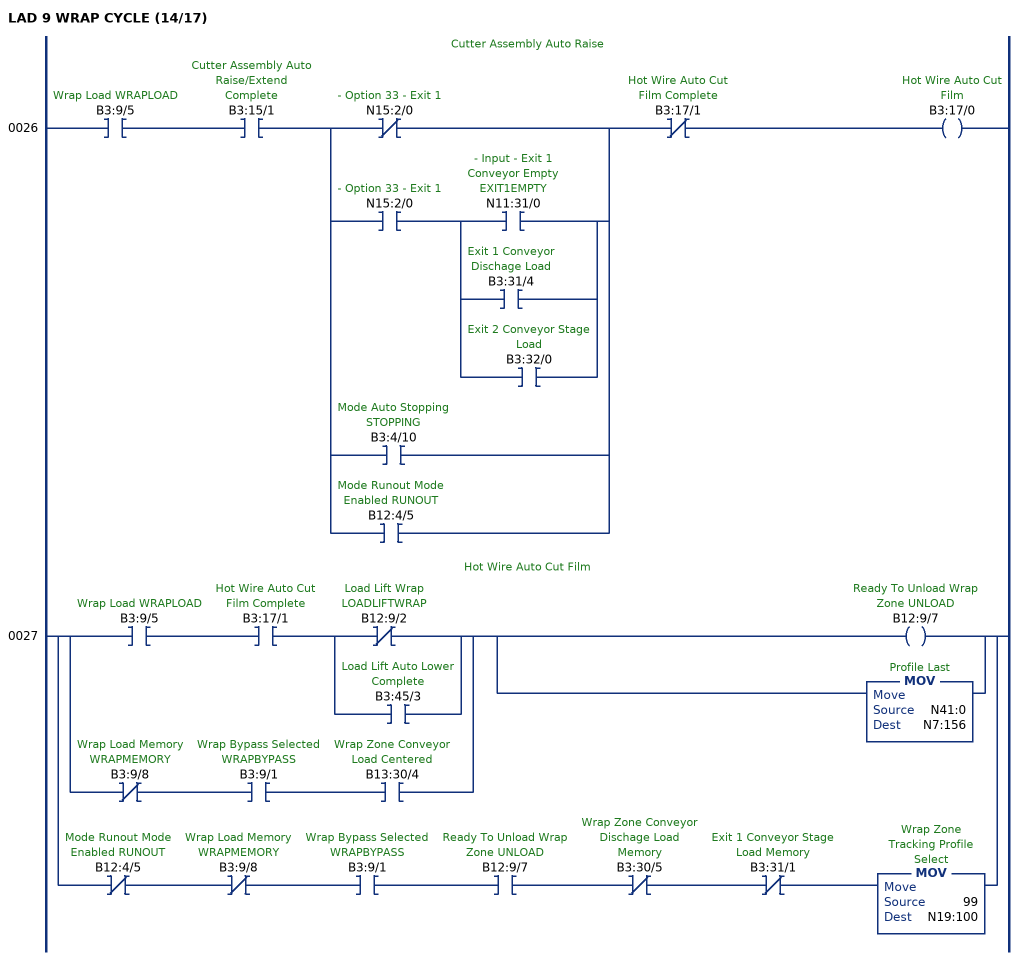
% Rung: 26 %
% Cutter Assembly Auto Raise %
SOR XIC B3:9/5 XIC B3:15/1 BST XIO N15:2/0 NXB XIC N15:2/0 BST XIC N11:31/0 NXB XIC B3:31/4 NXB XIC B3:32/0 BND NXB XIC B3:4/10 NXB XIC B12:4/5 BND XIO B3:17/1 OTE B3:17/0 EOR
%   B3:9/5  WRAPLOAD  "Wrap Load" %
%   B3:15/1  "Cutter Assembly Auto Raise/Extend Complete" %
%   N15:2/0  "- Option 33 - Exit 1" %
%   N11:31/0  EXIT1EMPTY  "- Input - Exit 1 Conveyor Empty" %
%   B3:31/4  "Exit 1 Conveyor Dischage Load" %
%   B3:32/0  "Exit 2 Conveyor Stage Load" %
%   B3:4/10  STOPPING  "Mode Auto Stopping" %
%   B12:4/5  RUNOUT  "Mode Runout Mode Enabled" %
%   B3:17/1  "Hot Wire Auto Cut Film Complete" %
%   B3:17/0  "Hot Wire Auto Cut Film" %
% Rung: 27 %
% Hot Wire Auto Cut Film %
SOR BST BST XIC B3:9/5 XIC B3:17/1 BST XIO B12:9/2 NXB XIC B3:45/3 BND NXB XIO B3:9/8 XIC B3:9/1 XIC B13:30/4 BND BST OTE B12:9/7 NXB MOV N41:0 N7:156 BND NXB XIO B12:4/5 XIO B3:9/8 XIC B3:9/1 XIC B12:9/7 XIO B3:30/5 XIO B3:31/1 MOV 99 N19:100 BND EOR
%   B3:9/5  WRAPLOAD  "Wrap Load" %
%   B3:17/1  "Hot Wire Auto Cut Film Complete" %
%   B12:9/2  LOADLIFTWRAP  "Load Lift Wrap" %
%   B3:45/3  "Load Lift Auto Lower Complete" %
%   B3:9/8  WRAPMEMORY  "Wrap Load Memory" %
%   B3:9/1  WRAPBYPASS  "Wrap Bypass Selected" %
%   B13:30/4  "Wrap Zone Conveyor Load Centered" %
%   B12:9/7  UNLOAD  "Ready To Unload Wrap Zone" %
%   N41:0  "Profile Max Index" %
%   N7:156  "Profile Last" %
%   B12:4/5  RUNOUT  "Mode Runout Mode Enabled" %
%   B3:30/5  "Wrap Zone Conveyor Dischage Load Memory" %
%   B3:31/1  "Exit 1 Conveyor Stage Load Memory" %
%   N19:100  "Wrap Zone Tracking Profile Select" %

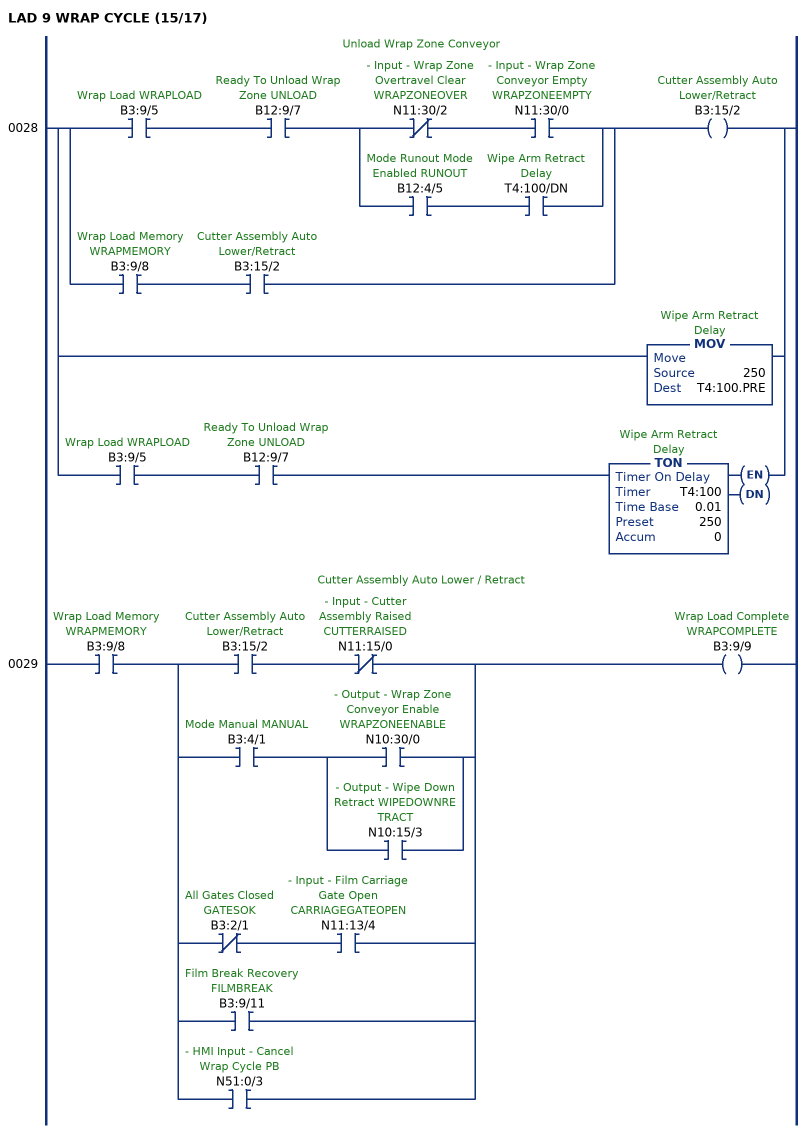
% Rung: 28 %
% Unload Wrap Zone Conveyor %
SOR BST BST XIC B3:9/5 XIC B12:9/7 BST XIO N11:30/2 XIC N11:30/0 NXB XIC B12:4/5 XIC T4:100/DN BND NXB XIC B3:9/8 XIC B3:15/2 BND OTE B3:15/2 NXB MOV 250 T4:100.PRE NXB XIC B3:9/5 XIC B12:9/7 TON T4:100 0.01 250 0 BND EOR
%   B3:9/5  WRAPLOAD  "Wrap Load" %
%   B12:9/7  UNLOAD  "Ready To Unload Wrap Zone" %
%   N11:30/2  WRAPZONEOVER  "- Input - Wrap Zone Overtravel Clear" %
%   N11:30/0  WRAPZONEEMPTY  "- Input - Wrap Zone Conveyor Empty" %
%   B12:4/5  RUNOUT  "Mode Runout Mode Enabled" %
%   T4:100  "Wipe Arm Retract Delay" %
%   B3:9/8  WRAPMEMORY  "Wrap Load Memory" %
%   B3:15/2  "Cutter Assembly Auto Lower/Retract" %
% Rung: 29 %
% Cutter Assembly Auto Lower / Retract %
SOR XIC B3:9/8 BST XIC B3:15/2 XIO N11:15/0 NXB XIC B3:4/1 BST XIC N10:30/0 NXB XIC N10:15/3 BND NXB XIO B3:2/1 XIC N11:13/4 NXB XIC B3:9/11 NXB XIC N51:0/3 BND OTE B3:9/9 EOR
%   B3:9/8  WRAPMEMORY  "Wrap Load Memory" %
%   B3:15/2  "Cutter Assembly Auto Lower/Retract" %
%   N11:15/0  CUTTERRAISED  "- Input - Cutter Assembly Raised" %
%   B3:4/1  MANUAL  "Mode Manual" %
%   N10:30/0  WRAPZONEENABLE  "- Output - Wrap Zone Conveyor Enable" %
%   N10:15/3  WIPEDOWNRETRACT  "- Output - Wipe Down Retract" %
%   B3:2/1  GATESOK  "All Gates Closed" %
%   N11:13/4  CARRIAGEGATEOPEN  "- Input - Film Carriage Gate Open" %
%   B3:9/11  FILMBREAK  "Film Break Recovery" %
%   N51:0/3  "- HMI Input - Cancel Wrap Cycle PB" %
%   B3:9/9  WRAPCOMPLETE  "Wrap Load Complete" %

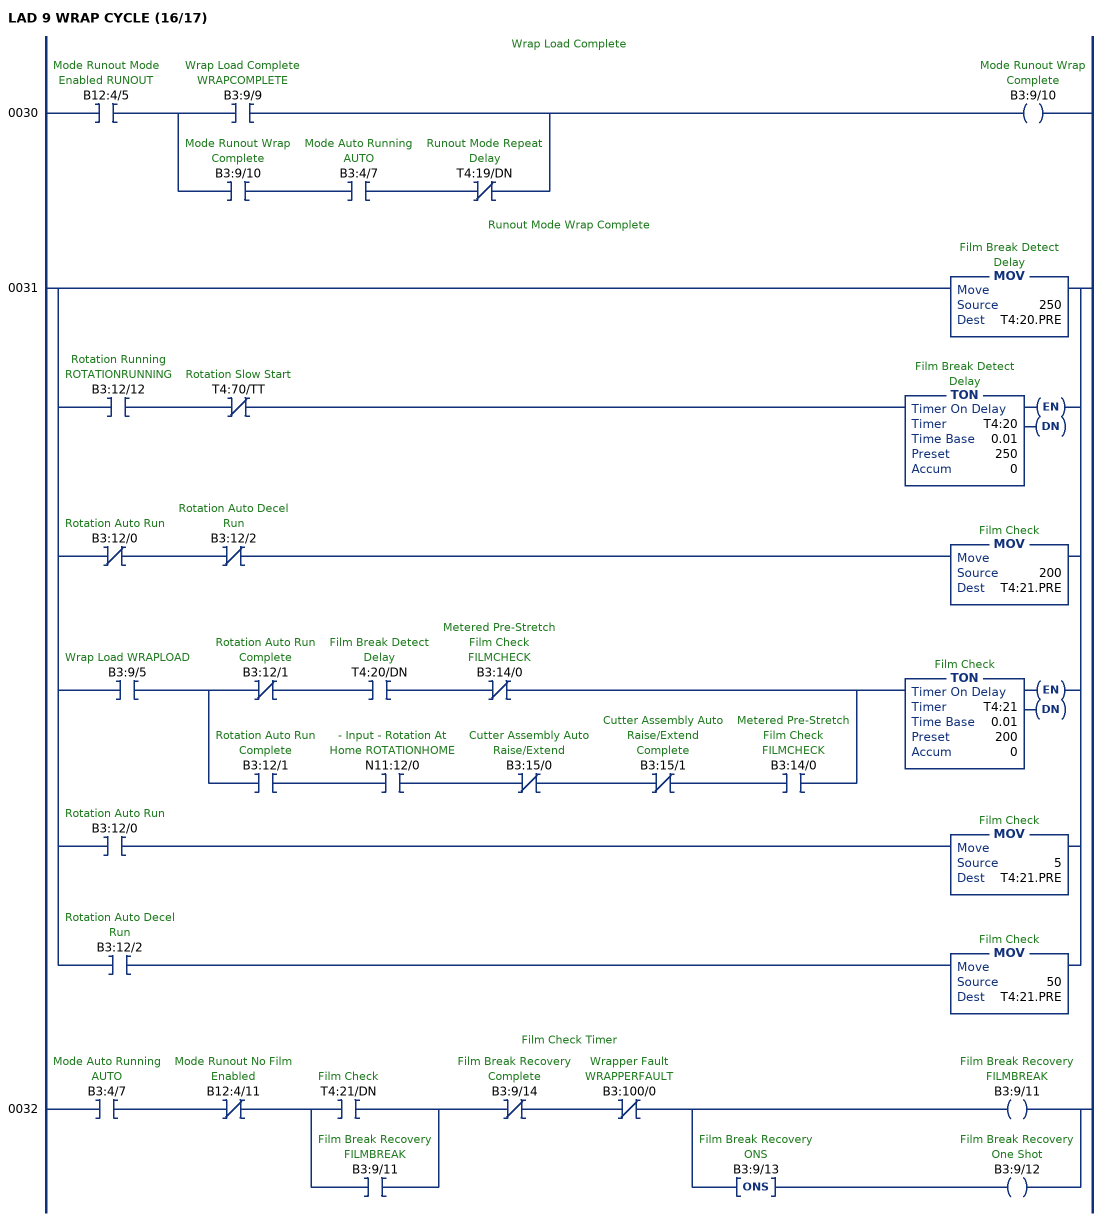
% Rung: 30 %
% Wrap Load Complete %
SOR XIC B12:4/5 BST XIC B3:9/9 NXB XIC B3:9/10 XIC B3:4/7 XIO T4:19/DN BND OTE B3:9/10 EOR
%   B12:4/5  RUNOUT  "Mode Runout Mode Enabled" %
%   B3:9/9  WRAPCOMPLETE  "Wrap Load Complete" %
%   B3:9/10  "Mode Runout Wrap Complete" %
%   B3:4/7  AUTO  "Mode Auto Running" %
%   T4:19  "Runout Mode Repeat Delay" %
% Rung: 31 %
% Runout Mode Wrap Complete %
SOR BST MOV 250 T4:20.PRE NXB XIC B3:12/12 XIO T4:70/TT TON T4:20 0.01 250 0 NXB XIO B3:12/0 XIO B3:12/2 MOV 200 T4:21.PRE NXB XIC B3:9/5 BST XIO B3:12/1 XIC T4:20/DN XIO B3:14/0 NXB XIC B3:12/1 XIC N11:12/0 XIO B3:15/0 XIO B3:15/1 XIC B3:14/0 BND TON T4:21 0.01 200 0 NXB BST XIC B3:12/0 MOV 5 T4:21.PRE NXB XIC B3:12/2 MOV 50 T4:21.PRE BND BND EOR
%   T4:20  "Film Break Detect Delay" %
%   B3:12/12  ROTATIONRUNNING  "Rotation Running" %
%   T4:70  "Rotation Slow Start" %
%   B3:12/0  "Rotation Auto Run" %
%   B3:12/2  "Rotation Auto Decel Run" %
%   T4:21  "Film Check" %
%   B3:9/5  WRAPLOAD  "Wrap Load" %
%   B3:12/1  "Rotation Auto Run Complete" %
%   B3:14/0  FILMCHECK  "Metered Pre-Stretch Film Check" %
%   N11:12/0  ROTATIONHOME  "- Input - Rotation At Home" %
%   B3:15/0  "Cutter Assembly Auto Raise/Extend" %
%   B3:15/1  "Cutter Assembly Auto Raise/Extend Complete" %
% Rung: 32 %
% Film Check Timer %
SOR XIC B3:4/7 XIO B12:4/11 BST XIC T4:21/DN NXB XIC B3:9/11 BND XIO B3:9/14 XIO B3:100/0 BST OTE B3:9/11 NXB ONS B3:9/13 OTE B3:9/12 BND EOR
%   B3:4/7  AUTO  "Mode Auto Running" %
%   B12:4/11  "Mode Runout No Film Enabled" %
%   T4:21  "Film Check" %
%   B3:9/11  FILMBREAK  "Film Break Recovery" %
%   B3:9/14  "Film Break Recovery Complete" %
%   B3:100/0  WRAPPERFAULT  "Wrapper Fault" %
%   B3:9/13  "Film Break Recovery ONS" %
%   B3:9/12  "Film Break Recovery One Shot" %

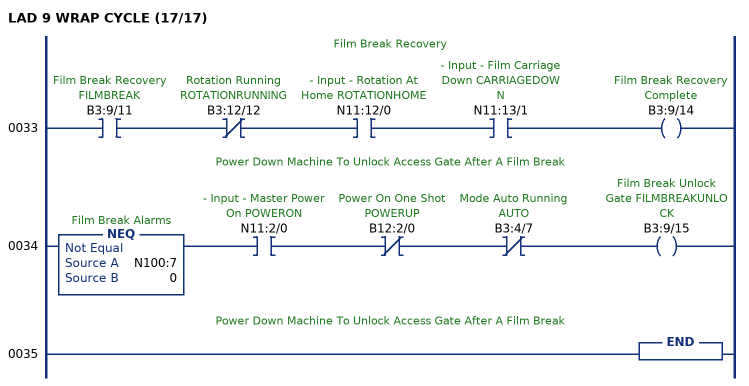
% Rung: 33 %
% Film Break Recovery %
SOR XIC B3:9/11 XIO B3:12/12 XIC N11:12/0 XIC N11:13/1 OTE B3:9/14 EOR
%   B3:9/11  FILMBREAK  "Film Break Recovery" %
%   B3:12/12  ROTATIONRUNNING  "Rotation Running" %
%   N11:12/0  ROTATIONHOME  "- Input - Rotation At Home" %
%   N11:13/1  CARRIAGEDOWN  "- Input - Film Carriage Down" %
%   B3:9/14  "Film Break Recovery Complete" %
% Rung: 34 %
% Power Down Machine To Unlock Access Gate After A Film Break %
SOR NEQ N100:7 0 XIC N11:2/0 XIO B12:2/0 XIO B3:4/7 OTE B3:9/15 EOR
%   N100:7  "Film Break Alarms" %
%   N11:2/0  POWERON  "- Input - Master Power On" %
%   B12:2/0  POWERUP  "Power On One Shot" %
%   B3:4/7  AUTO  "Mode Auto Running" %
%   B3:9/15  FILMBREAKUNLOCK  "Film Break Unlock Gate" %
% Rung: 35 %
% Power Down Machine To Unlock Access Gate After A Film Break %
SOR END EOR

LADDER 10 "OUTPUTS"
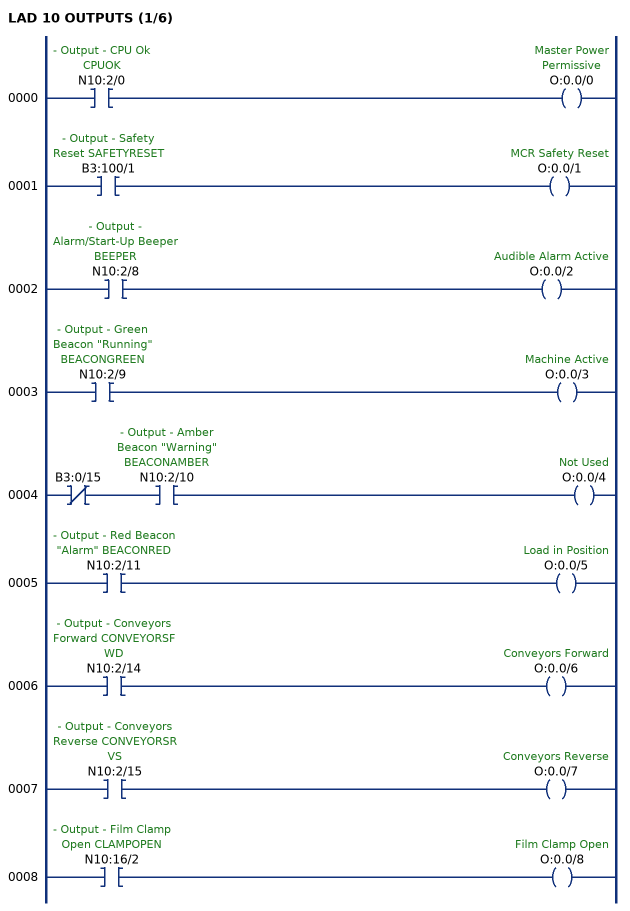
% Rung: 0 %
SOR XIC N10:2/0 OTE O:0.0/0 EOR
%   N10:2/0  CPUOK  "- Output - CPU Ok" %
%   O:0.0/0  "Master Power Permissive" %
% Rung: 1 %
SOR XIC B3:100/1 OTE O:0.0/1 EOR
%   B3:100/1  SAFETYRESET  "- Output - Safety Reset" %
%   O:0.0/1  "MCR Safety Reset" %
% Rung: 2 %
SOR XIC N10:2/8 OTE O:0.0/2 EOR
%   N10:2/8  BEEPER  "- Output - Alarm/Start-Up Beeper" %
%   O:0.0/2  "Audible Alarm Active" %
% Rung: 3 %
SOR XIC N10:2/9 OTE O:0.0/3 EOR
%   N10:2/9  BEACONGREEN  "- Output - Green Beacon "Running"" %
%   O:0.0/3  "Machine Active" %
% Rung: 4 %
SOR XIO B3:0/15 XIC N10:2/10 OTE O:0.0/4 EOR
%   N10:2/10  BEACONAMBER  "- Output - Amber Beacon "Warning"" %
%   O:0.0/4  "Not Used" %
% Rung: 5 %
SOR XIC N10:2/11 OTE O:0.0/5 EOR
%   N10:2/11  BEACONRED  "- Output - Red Beacon "Alarm"" %
%   O:0.0/5  "Load in Position" %
% Rung: 6 %
SOR XIC N10:2/14 OTE O:0.0/6 EOR
%   N10:2/14  CONVEYORSFWD  "- Output - Conveyors Forward" %
%   O:0.0/6  "Conveyors Forward" %
% Rung: 7 %
SOR XIC N10:2/15 OTE O:0.0/7 EOR
%   N10:2/15  CONVEYORSRVS  "- Output - Conveyors Reverse" %
%   O:0.0/7  "Conveyors Reverse" %
% Rung: 8 %
SOR XIC N10:16/2 OTE O:0.0/8 EOR
%   N10:16/2  CLAMPOPEN  "- Output - Film Clamp Open" %
%   O:0.0/8  "Film Clamp Open" %

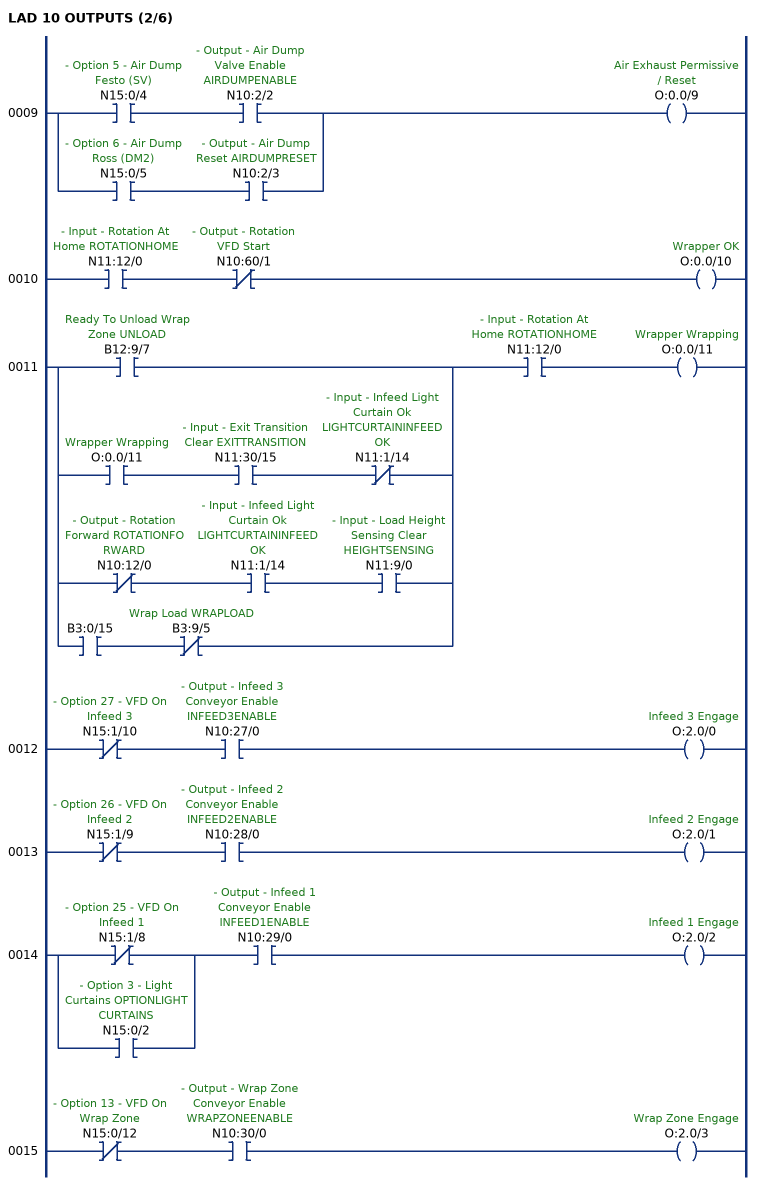
% Rung: 9 %
SOR BST XIC N15:0/4 XIC N10:2/2 NXB XIC N15:0/5 XIC N10:2/3 BND OTE O:0.0/9 EOR
%   N15:0/4  "- Option 5 - Air Dump Festo (SV)" %
%   N10:2/2  AIRDUMPENABLE  "- Output - Air Dump Valve Enable" %
%   N15:0/5  "- Option 6 - Air Dump Ross (DM2)" %
%   N10:2/3  AIRDUMPRESET  "- Output - Air Dump Reset" %
%   O:0.0/9  "Air Exhaust Permissive / Reset" %
% Rung: 10 %
SOR XIC N11:12/0 XIO N10:60/1 OTE O:0.0/10 EOR
%   N11:12/0  ROTATIONHOME  "- Input - Rotation At Home" %
%   N10:60/1  "- Output - Rotation VFD Start" %
%   O:0.0/10  "Wrapper OK" %
% Rung: 11 %
SOR BST XIC B12:9/7 NXB BST XIC O:0.0/11 XIC N11:30/15 XIO N11:1/14 NXB XIO N10:12/0 XIC N11:1/14 XIC N11:9/0 BND NXB XIC B3:0/15 XIO B3:9/5 BND XIC N11:12/0 OTE O:0.0/11 EOR
%   B12:9/7  UNLOAD  "Ready To Unload Wrap Zone" %
%   O:0.0/11  "Wrapper Wrapping" %
%   N11:30/15  EXITTRANSITION  "- Input - Exit Transition Clear" %
%   N11:1/14  LIGHTCURTAININFEEDOK  "- Input - Infeed Light Curtain Ok" %
%   N10:12/0  ROTATIONFORWARD  "- Output - Rotation Forward" %
%   N11:9/0  HEIGHTSENSING  "- Input - Load Height Sensing Clear" %
%   B3:9/5  WRAPLOAD  "Wrap Load" %
%   N11:12/0  ROTATIONHOME  "- Input - Rotation At Home" %
% Rung: 12 %
SOR XIO N15:1/10 XIC N10:27/0 OTE O:2.0/0 EOR
%   N15:1/10  "- Option 27 - VFD On Infeed 3" %
%   N10:27/0  INFEED3ENABLE  "- Output - Infeed 3 Conveyor Enable" %
%   O:2.0/0  "Infeed 3 Engage" %
% Rung: 13 %
SOR XIO N15:1/9 XIC N10:28/0 OTE O:2.0/1 EOR
%   N15:1/9  "- Option 26 - VFD On Infeed 2" %
%   N10:28/0  INFEED2ENABLE  "- Output - Infeed 2 Conveyor Enable" %
%   O:2.0/1  "Infeed 2 Engage" %
% Rung: 14 %
SOR BST XIO N15:1/8 NXB XIC N15:0/2 BND XIC N10:29/0 OTE O:2.0/2 EOR
%   N15:1/8  "- Option 25 - VFD On Infeed 1" %
%   N15:0/2  OPTIONLIGHTCURTAINS  "- Option 3 - Light Curtains" %
%   N10:29/0  INFEED1ENABLE  "- Output - Infeed 1 Conveyor Enable" %
%   O:2.0/2  "Infeed 1 Engage" %
% Rung: 15 %
SOR XIO N15:0/12 XIC N10:30/0 OTE O:2.0/3 EOR
%   N15:0/12  "- Option 13 - VFD On Wrap Zone" %
%   N10:30/0  WRAPZONEENABLE  "- Output - Wrap Zone Conveyor Enable" %
%   O:2.0/3  "Wrap Zone Engage" %

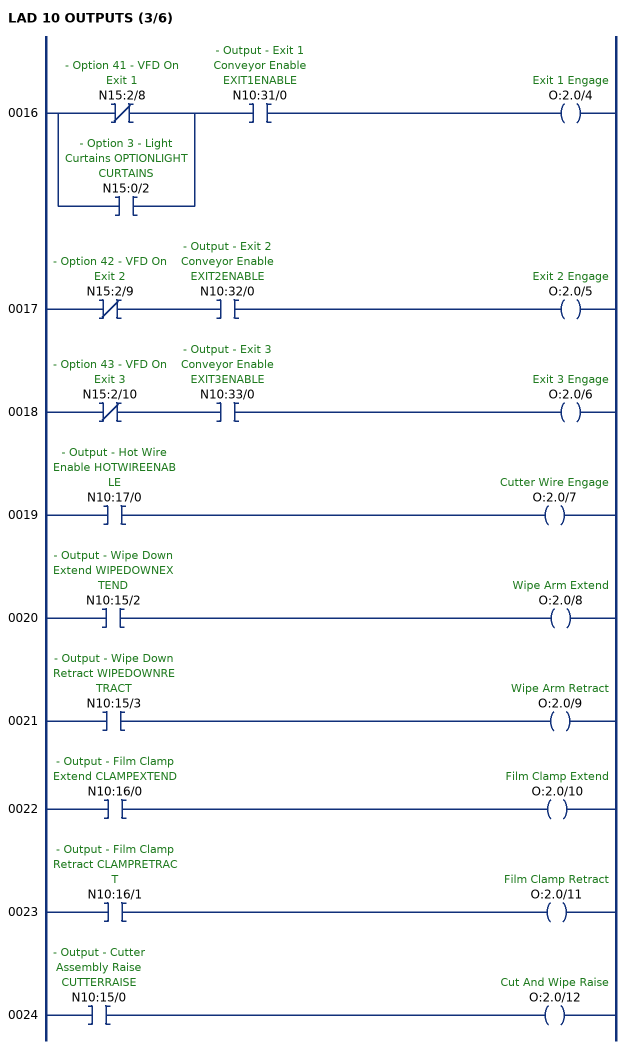
% Rung: 16 %
SOR BST XIO N15:2/8 NXB XIC N15:0/2 BND XIC N10:31/0 OTE O:2.0/4 EOR
%   N15:2/8  "- Option 41 - VFD On Exit 1" %
%   N15:0/2  OPTIONLIGHTCURTAINS  "- Option 3 - Light Curtains" %
%   N10:31/0  EXIT1ENABLE  "- Output - Exit 1 Conveyor Enable" %
%   O:2.0/4  "Exit 1 Engage" %
% Rung: 17 %
SOR XIO N15:2/9 XIC N10:32/0 OTE O:2.0/5 EOR
%   N15:2/9  "- Option 42 - VFD On Exit 2" %
%   N10:32/0  EXIT2ENABLE  "- Output - Exit 2 Conveyor Enable" %
%   O:2.0/5  "Exit 2 Engage" %
% Rung: 18 %
SOR XIO N15:2/10 XIC N10:33/0 OTE O:2.0/6 EOR
%   N15:2/10  "- Option 43 - VFD On Exit 3" %
%   N10:33/0  EXIT3ENABLE  "- Output - Exit 3 Conveyor Enable" %
%   O:2.0/6  "Exit 3 Engage" %
% Rung: 19 %
SOR XIC N10:17/0 OTE O:2.0/7 EOR
%   N10:17/0  HOTWIREENABLE  "- Output - Hot Wire Enable" %
%   O:2.0/7  "Cutter Wire Engage" %
% Rung: 20 %
SOR XIC N10:15/2 OTE O:2.0/8 EOR
%   N10:15/2  WIPEDOWNEXTEND  "- Output - Wipe Down Extend" %
%   O:2.0/8  "Wipe Arm Extend" %
% Rung: 21 %
SOR XIC N10:15/3 OTE O:2.0/9 EOR
%   N10:15/3  WIPEDOWNRETRACT  "- Output - Wipe Down Retract" %
%   O:2.0/9  "Wipe Arm Retract" %
% Rung: 22 %
SOR XIC N10:16/0 OTE O:2.0/10 EOR
%   N10:16/0  CLAMPEXTEND  "- Output - Film Clamp Extend" %
%   O:2.0/10  "Film Clamp Extend" %
% Rung: 23 %
SOR XIC N10:16/1 OTE O:2.0/11 EOR
%   N10:16/1  CLAMPRETRACT  "- Output - Film Clamp Retract" %
%   O:2.0/11  "Film Clamp Retract" %
% Rung: 24 %
SOR XIC N10:15/0 OTE O:2.0/12 EOR
%   N10:15/0  CUTTERRAISE  "- Output - Cutter Assembly Raise" %
%   O:2.0/12  "Cut And Wipe Raise" %

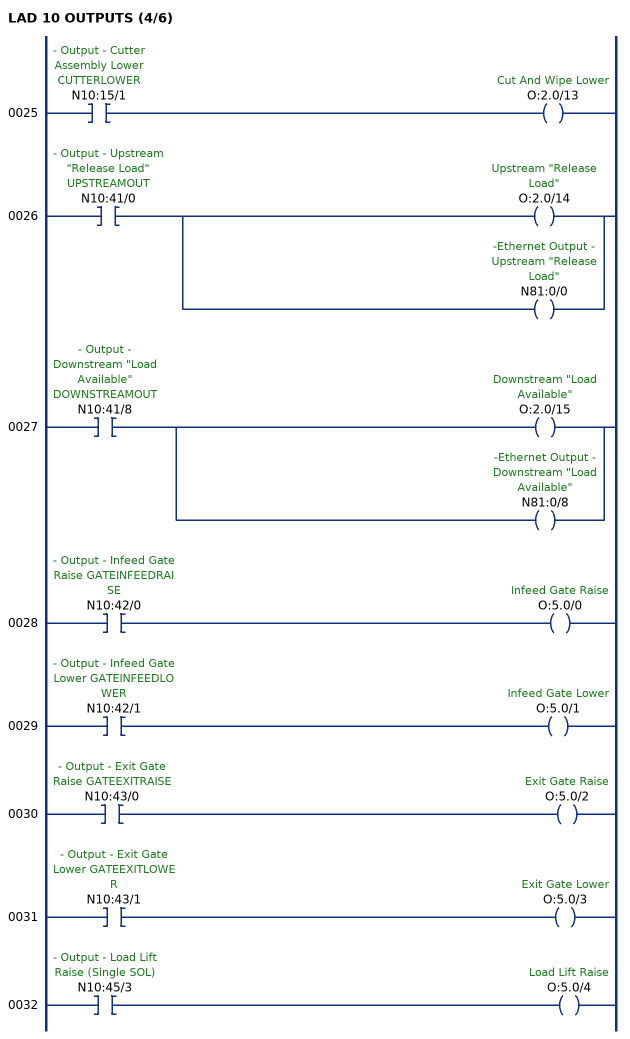
% Rung: 25 %
SOR XIC N10:15/1 OTE O:2.0/13 EOR
%   N10:15/1  CUTTERLOWER  "- Output - Cutter Assembly Lower" %
%   O:2.0/13  "Cut And Wipe Lower" %
% Rung: 26 %
SOR XIC N10:41/0 BST OTE O:2.0/14 NXB OTE N81:0/0 BND EOR
%   N10:41/0  UPSTREAMOUT  "- Output - Upstream "Release Load"" %
%   O:2.0/14  "Upstream "Release Load"" %
%   N81:0/0  "-Ethernet Output - Upstream "Release Load"" %
% Rung: 27 %
SOR XIC N10:41/8 BST OTE O:2.0/15 NXB OTE N81:0/8 BND EOR
%   N10:41/8  DOWNSTREAMOUT  "- Output - Downstream "Load Available"" %
%   O:2.0/15  "Downstream "Load Available"" %
%   N81:0/8  "-Ethernet Output - Downstream "Load Available"" %
% Rung: 28 %
SOR XIC N10:42/0 OTE O:5.0/0 EOR
%   N10:42/0  GATEINFEEDRAISE  "- Output - Infeed Gate Raise" %
%   O:5.0/0  "Infeed Gate Raise" %
% Rung: 29 %
SOR XIC N10:42/1 OTE O:5.0/1 EOR
%   N10:42/1  GATEINFEEDLOWER  "- Output - Infeed Gate Lower" %
%   O:5.0/1  "Infeed Gate Lower" %
% Rung: 30 %
SOR XIC N10:43/0 OTE O:5.0/2 EOR
%   N10:43/0  GATEEXITRAISE  "- Output - Exit Gate Raise" %
%   O:5.0/2  "Exit Gate Raise" %
% Rung: 31 %
SOR XIC N10:43/1 OTE O:5.0/3 EOR
%   N10:43/1  GATEEXITLOWER  "- Output - Exit Gate Lower" %
%   O:5.0/3  "Exit Gate Lower" %
% Rung: 32 %
SOR XIC N10:45/3 OTE O:5.0/4 EOR
%   N10:45/3  "- Output - Load Lift Raise (Single SOL)" %
%   O:5.0/4  "Load Lift Raise" %

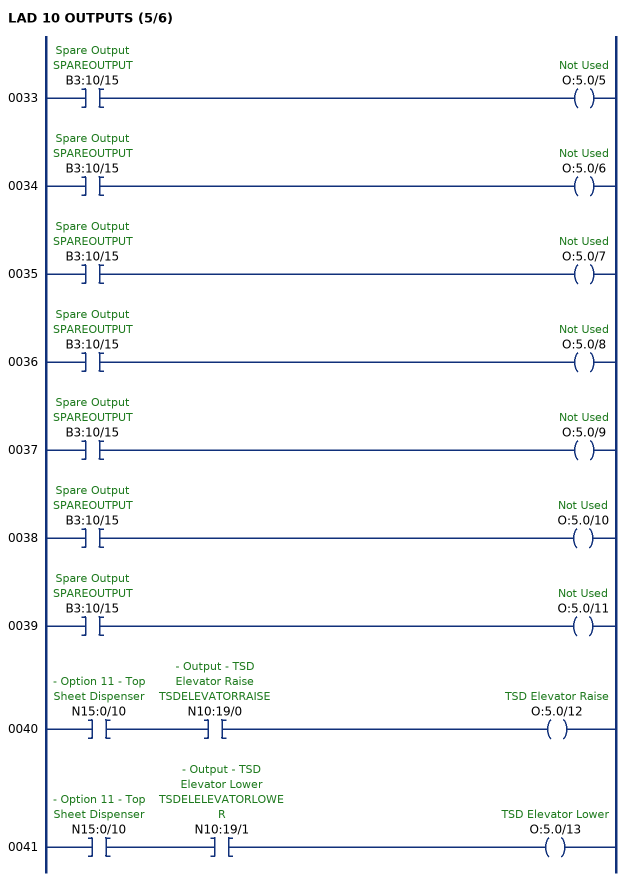
% Rung: 33 %
SOR XIC B3:10/15 OTE O:5.0/5 EOR
%   B3:10/15  SPAREOUTPUT  "Spare Output" %
%   O:5.0/5  "Not Used" %
% Rung: 34 %
SOR XIC B3:10/15 OTE O:5.0/6 EOR
%   B3:10/15  SPAREOUTPUT  "Spare Output" %
%   O:5.0/6  "Not Used" %
% Rung: 35 %
SOR XIC B3:10/15 OTE O:5.0/7 EOR
%   B3:10/15  SPAREOUTPUT  "Spare Output" %
%   O:5.0/7  "Not Used" %
% Rung: 36 %
SOR XIC B3:10/15 OTE O:5.0/8 EOR
%   B3:10/15  SPAREOUTPUT  "Spare Output" %
%   O:5.0/8  "Not Used" %
% Rung: 37 %
SOR XIC B3:10/15 OTE O:5.0/9 EOR
%   B3:10/15  SPAREOUTPUT  "Spare Output" %
%   O:5.0/9  "Not Used" %
% Rung: 38 %
SOR XIC B3:10/15 OTE O:5.0/10 EOR
%   B3:10/15  SPAREOUTPUT  "Spare Output" %
%   O:5.0/10  "Not Used" %
% Rung: 39 %
SOR XIC B3:10/15 OTE O:5.0/11 EOR
%   B3:10/15  SPAREOUTPUT  "Spare Output" %
%   O:5.0/11  "Not Used" %
% Rung: 40 %
SOR XIC N15:0/10 XIC N10:19/0 OTE O:5.0/12 EOR
%   N15:0/10  "- Option 11 - Top Sheet Dispenser" %
%   N10:19/0  TSDELEVATORRAISE  "- Output - TSD Elevator Raise" %
%   O:5.0/12  "TSD Elevator Raise" %
% Rung: 41 %
SOR XIC N15:0/10 XIC N10:19/1 OTE O:5.0/13 EOR
%   N15:0/10  "- Option 11 - Top Sheet Dispenser" %
%   N10:19/1  TSDELELEVATORLOWER  "- Output - TSD Elevator Lower" %
%   O:5.0/13  "TSD Elevator Lower" %

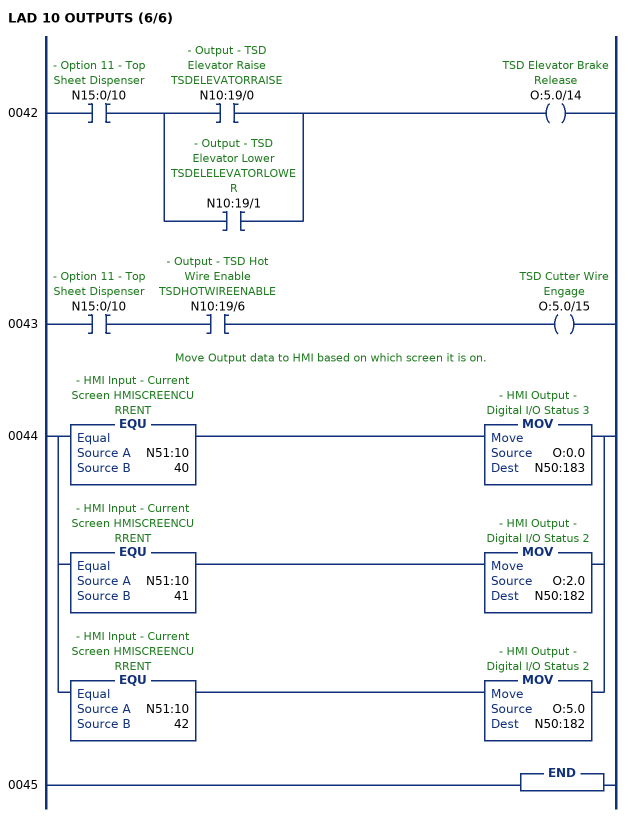
% Rung: 42 %
SOR XIC N15:0/10 BST XIC N10:19/0 NXB XIC N10:19/1 BND OTE O:5.0/14 EOR
%   N15:0/10  "- Option 11 - Top Sheet Dispenser" %
%   N10:19/0  TSDELEVATORRAISE  "- Output - TSD Elevator Raise" %
%   N10:19/1  TSDELELEVATORLOWER  "- Output - TSD Elevator Lower" %
%   O:5.0/14  "TSD Elevator Brake Release" %
% Rung: 43 %
SOR XIC N15:0/10 XIC N10:19/6 OTE O:5.0/15 EOR
%   N15:0/10  "- Option 11 - Top Sheet Dispenser" %
%   N10:19/6  TSDHOTWIREENABLE  "- Output - TSD Hot Wire Enable" %
%   O:5.0/15  "TSD Cutter Wire Engage" %
% Rung: 44 %
% Move Output data to HMI based on which screen it is on. %
SOR BST EQU N51:10 40 MOV O:0.0 N50:183 NXB EQU N51:10 41 MOV O:2.0 N50:182 NXB EQU N51:10 42 MOV O:5.0 N50:182 BND EOR
%   N51:10  HMISCREENCURRENT  "- HMI Input - Current Screen" %
%   N50:183  "- HMI Output - Digital I/O Status 3" %
%   N50:182  "- HMI Output - Digital I/O Status 2" %
% Rung: 45 %
SOR END EOR

LADDER 11 "INPUTS"
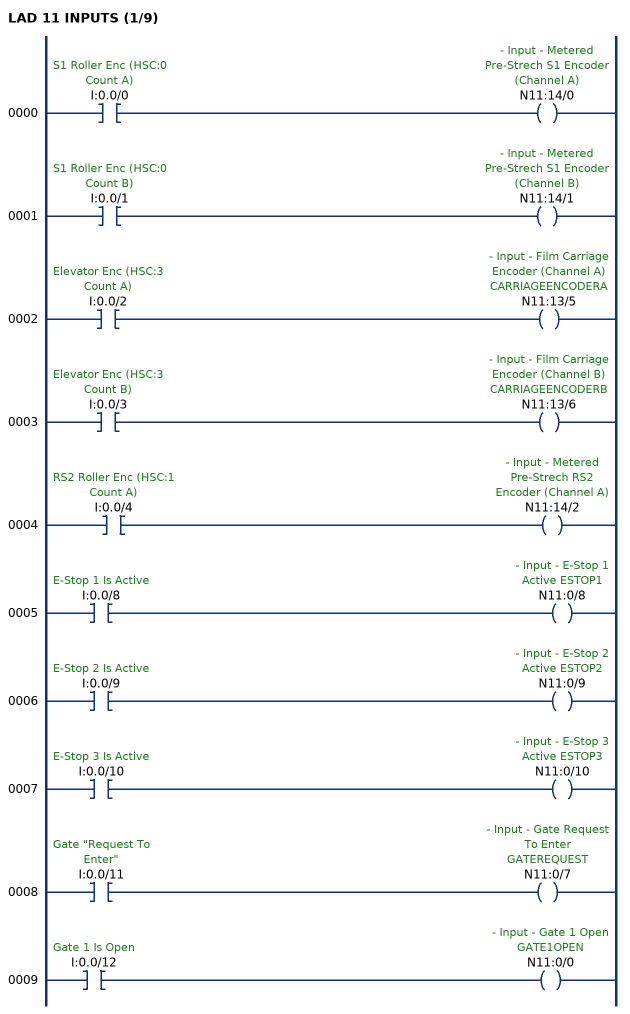
% Rung: 0 %
SOR XIC I:0.0/0 OTE N11:14/0 EOR
%   I:0.0/0  "S1 Roller Enc (HSC:0 Count A)" %
%   N11:14/0  "- Input - Metered Pre-Strech S1 Encoder (Channel A)" %
% Rung: 1 %
SOR XIC I:0.0/1 OTE N11:14/1 EOR
%   I:0.0/1  "S1 Roller Enc (HSC:0 Count B)" %
%   N11:14/1  "- Input - Metered Pre-Strech S1 Encoder (Channel B)" %
% Rung: 2 %
SOR XIC I:0.0/2 OTE N11:13/5 EOR
%   I:0.0/2  "Elevator Enc (HSC:3 Count A)" %
%   N11:13/5  CARRIAGEENCODERA  "- Input - Film Carriage Encoder (Channel A)" %
% Rung: 3 %
SOR XIC I:0.0/3 OTE N11:13/6 EOR
%   I:0.0/3  "Elevator Enc (HSC:3 Count B)" %
%   N11:13/6  CARRIAGEENCODERB  "- Input - Film Carriage Encoder (Channel B)" %
% Rung: 4 %
SOR XIC I:0.0/4 OTE N11:14/2 EOR
%   I:0.0/4  "RS2 Roller Enc (HSC:1 Count A)" %
%   N11:14/2  "- Input - Metered Pre-Strech RS2 Encoder (Channel A)" %
% Rung: 5 %
SOR XIC I:0.0/8 OTE N11:0/8 EOR
%   I:0.0/8  "E-Stop 1 Is Active" %
%   N11:0/8  ESTOP1  "- Input - E-Stop 1 Active" %
% Rung: 6 %
SOR XIC I:0.0/9 OTE N11:0/9 EOR
%   I:0.0/9  "E-Stop 2 Is Active" %
%   N11:0/9  ESTOP2  "- Input - E-Stop 2 Active" %
% Rung: 7 %
SOR XIC I:0.0/10 OTE N11:0/10 EOR
%   I:0.0/10  "E-Stop 3 Is Active" %
%   N11:0/10  ESTOP3  "- Input - E-Stop 3 Active" %
% Rung: 8 %
SOR XIC I:0.0/11 OTE N11:0/7 EOR
%   I:0.0/11  "Gate "Request To Enter"" %
%   N11:0/7  GATEREQUEST  "- Input - Gate Request To Enter" %
% Rung: 9 %
SOR XIC I:0.0/12 OTE N11:0/0 EOR
%   I:0.0/12  "Gate 1 Is Open" %
%   N11:0/0  GATE1OPEN  "- Input - Gate 1 Open" %

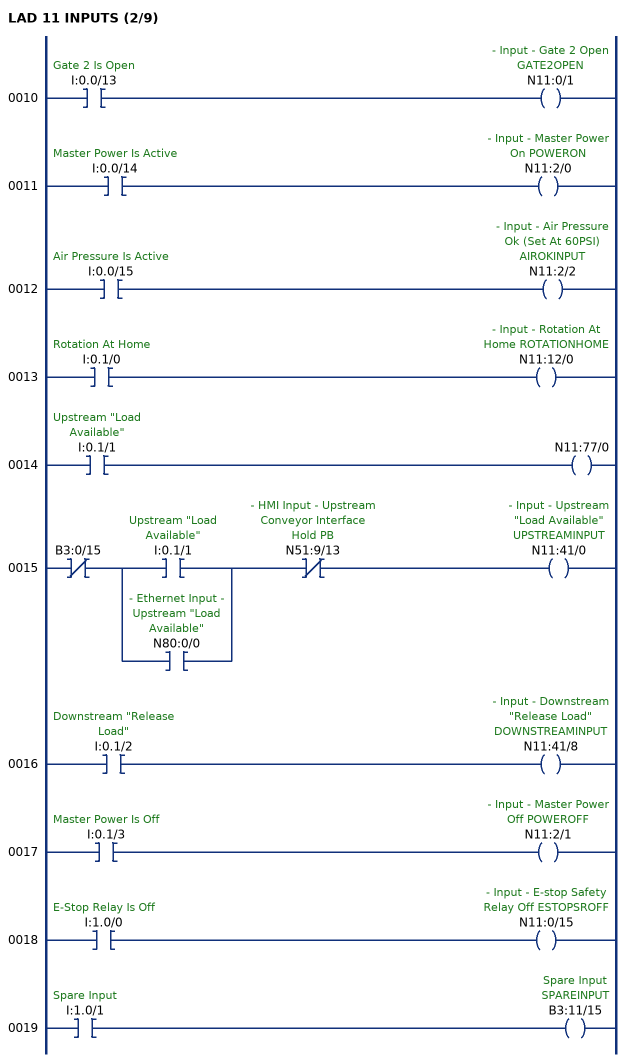
% Rung: 10 %
SOR XIC I:0.0/13 OTE N11:0/1 EOR
%   I:0.0/13  "Gate 2 Is Open" %
%   N11:0/1  GATE2OPEN  "- Input - Gate 2 Open" %
% Rung: 11 %
SOR XIC I:0.0/14 OTE N11:2/0 EOR
%   I:0.0/14  "Master Power Is Active" %
%   N11:2/0  POWERON  "- Input - Master Power On" %
% Rung: 12 %
SOR XIC I:0.0/15 OTE N11:2/2 EOR
%   I:0.0/15  "Air Pressure Is Active" %
%   N11:2/2  AIROKINPUT  "- Input - Air Pressure Ok (Set At 60PSI)" %
% Rung: 13 %
SOR XIC I:0.1/0 OTE N11:12/0 EOR
%   I:0.1/0  "Rotation At Home" %
%   N11:12/0  ROTATIONHOME  "- Input - Rotation At Home" %
% Rung: 14 %
SOR XIC I:0.1/1 OTE N11:77/0 EOR
%   I:0.1/1  "Upstream "Load Available"" %
% Rung: 15 %
SOR XIO B3:0/15 BST XIC I:0.1/1 NXB XIC N80:0/0 BND XIO N51:9/13 OTE N11:41/0 EOR
%   I:0.1/1  "Upstream "Load Available"" %
%   N80:0/0  "- Ethernet Input - Upstream "Load Available"" %
%   N51:9/13  "- HMI Input - Upstream Conveyor Interface Hold PB" %
%   N11:41/0  UPSTREAMINPUT  "- Input - Upstream "Load Available"" %
% Rung: 16 %
SOR XIC I:0.1/2 OTE N11:41/8 EOR
%   I:0.1/2  "Downstream "Release Load"" %
%   N11:41/8  DOWNSTREAMINPUT  "- Input - Downstream "Release Load"" %
% Rung: 17 %
SOR XIC I:0.1/3 OTE N11:2/1 EOR
%   I:0.1/3  "Master Power Is Off" %
%   N11:2/1  POWEROFF  "- Input - Master Power Off" %
% Rung: 18 %
SOR XIC I:1.0/0 OTE N11:0/15 EOR
%   I:1.0/0  "E-Stop Relay Is Off" %
%   N11:0/15  ESTOPSROFF  "- Input - E-stop Safety Relay Off" %
% Rung: 19 %
SOR XIC I:1.0/1 OTE B3:11/15 EOR
%   I:1.0/1  "Spare Input" %
%   B3:11/15  SPAREINPUT  "Spare Input" %

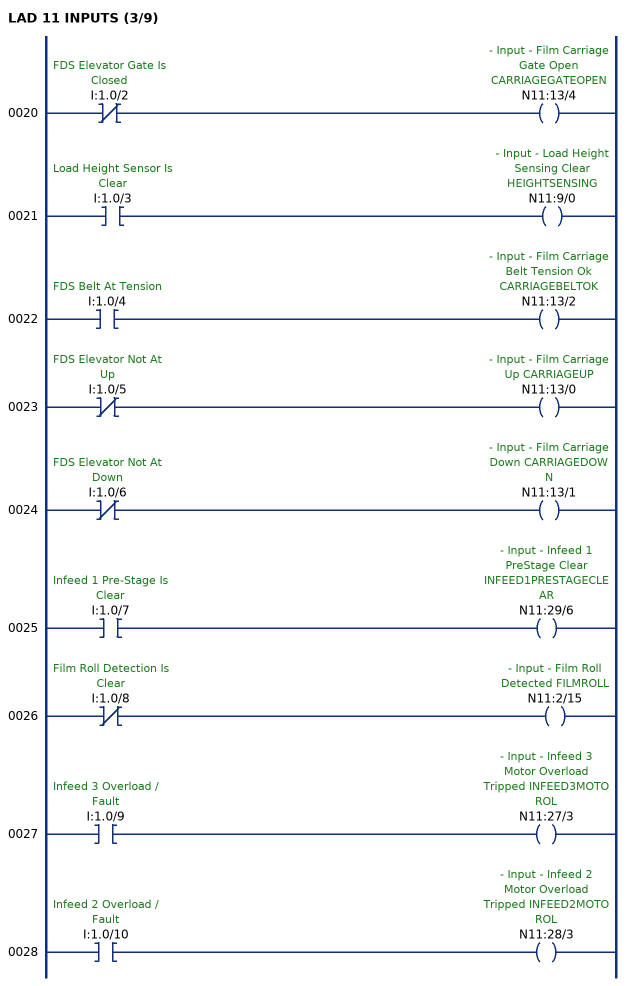
% Rung: 20 %
SOR XIO I:1.0/2 OTE N11:13/4 EOR
%   I:1.0/2  "FDS Elevator Gate Is Closed" %
%   N11:13/4  CARRIAGEGATEOPEN  "- Input - Film Carriage Gate Open" %
% Rung: 21 %
SOR XIC I:1.0/3 OTE N11:9/0 EOR
%   I:1.0/3  "Load Height Sensor Is Clear" %
%   N11:9/0  HEIGHTSENSING  "- Input - Load Height Sensing Clear" %
% Rung: 22 %
SOR XIC I:1.0/4 OTE N11:13/2 EOR
%   I:1.0/4  "FDS Belt At Tension" %
%   N11:13/2  CARRIAGEBELTOK  "- Input - Film Carriage Belt Tension Ok" %
% Rung: 23 %
SOR XIO I:1.0/5 OTE N11:13/0 EOR
%   I:1.0/5  "FDS Elevator Not At Up" %
%   N11:13/0  CARRIAGEUP  "- Input - Film Carriage Up" %
% Rung: 24 %
SOR XIO I:1.0/6 OTE N11:13/1 EOR
%   I:1.0/6  "FDS Elevator Not At Down" %
%   N11:13/1  CARRIAGEDOWN  "- Input - Film Carriage Down" %
% Rung: 25 %
SOR XIC I:1.0/7 OTE N11:29/6 EOR
%   I:1.0/7  "Infeed 1 Pre-Stage Is Clear" %
%   N11:29/6  INFEED1PRESTAGECLEAR  "- Input - Infeed 1 PreStage Clear" %
% Rung: 26 %
SOR XIO I:1.0/8 OTE N11:2/15 EOR
%   I:1.0/8  "Film Roll Detection Is Clear" %
%   N11:2/15  FILMROLL  "- Input - Film Roll Detected" %
% Rung: 27 %
SOR XIC I:1.0/9 OTE N11:27/3 EOR
%   I:1.0/9  "Infeed 3 Overload / Fault" %
%   N11:27/3  INFEED3MOTOROL  "- Input - Infeed 3 Motor Overload Tripped" %
% Rung: 28 %
SOR XIC I:1.0/10 OTE N11:28/3 EOR
%   I:1.0/10  "Infeed 2 Overload / Fault" %
%   N11:28/3  INFEED2MOTOROL  "- Input - Infeed 2 Motor Overload Tripped" %

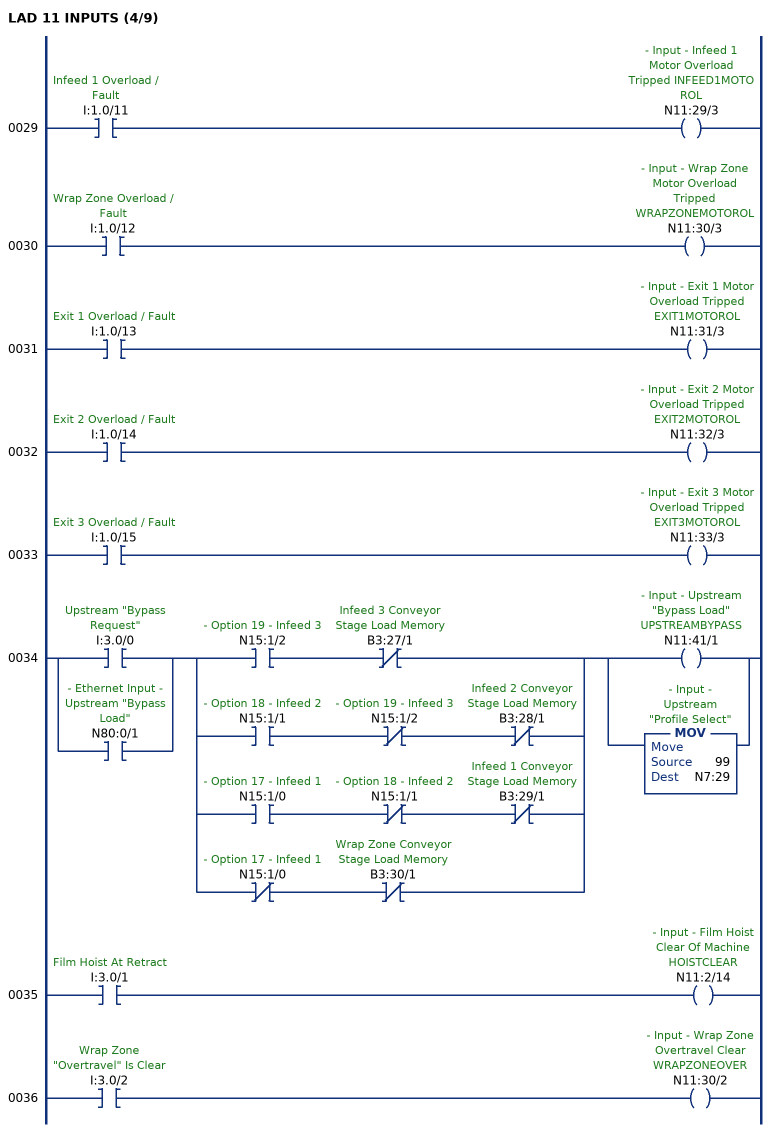
% Rung: 29 %
SOR XIC I:1.0/11 OTE N11:29/3 EOR
%   I:1.0/11  "Infeed 1 Overload / Fault" %
%   N11:29/3  INFEED1MOTOROL  "- Input - Infeed 1 Motor Overload Tripped" %
% Rung: 30 %
SOR XIC I:1.0/12 OTE N11:30/3 EOR
%   I:1.0/12  "Wrap Zone Overload / Fault" %
%   N11:30/3  WRAPZONEMOTOROL  "- Input - Wrap Zone Motor Overload Tripped" %
% Rung: 31 %
SOR XIC I:1.0/13 OTE N11:31/3 EOR
%   I:1.0/13  "Exit 1 Overload / Fault" %
%   N11:31/3  EXIT1MOTOROL  "- Input - Exit 1 Motor Overload Tripped" %
% Rung: 32 %
SOR XIC I:1.0/14 OTE N11:32/3 EOR
%   I:1.0/14  "Exit 2 Overload / Fault" %
%   N11:32/3  EXIT2MOTOROL  "- Input - Exit 2 Motor Overload Tripped" %
% Rung: 33 %
SOR XIC I:1.0/15 OTE N11:33/3 EOR
%   I:1.0/15  "Exit 3 Overload / Fault" %
%   N11:33/3  EXIT3MOTOROL  "- Input - Exit 3 Motor Overload Tripped" %
% Rung: 34 %
SOR BST XIC I:3.0/0 NXB XIC N80:0/1 BND BST XIC N15:1/2 XIO B3:27/1 NXB XIC N15:1/1 XIO N15:1/2 XIO B3:28/1 NXB XIC N15:1/0 XIO N15:1/1 XIO B3:29/1 NXB XIO N15:1/0 XIO B3:30/1 BND BST OTE N11:41/1 NXB MOV 99 N7:29 BND EOR
%   I:3.0/0  "Upstream "Bypass Request"" %
%   N80:0/1  "- Ethernet Input - Upstream "Bypass Load"" %
%   N15:1/2  "- Option 19 - Infeed 3" %
%   B3:27/1  "Infeed 3 Conveyor Stage Load Memory" %
%   N15:1/1  "- Option 18 - Infeed 2" %
%   B3:28/1  "Infeed 2 Conveyor Stage Load Memory" %
%   N15:1/0  "- Option 17 - Infeed 1" %
%   B3:29/1  "Infeed 1 Conveyor Stage Load Memory" %
%   B3:30/1  "Wrap Zone Conveyor Stage Load Memory" %
%   N11:41/1  UPSTREAMBYPASS  "- Input - Upstream "Bypass Load"" %
%   N7:29  "- Input - Upstream "Profile Select"" %
% Rung: 35 %
SOR XIC I:3.0/1 OTE N11:2/14 EOR
%   I:3.0/1  "Film Hoist At Retract" %
%   N11:2/14  HOISTCLEAR  "- Input - Film Hoist Clear Of Machine" %
% Rung: 36 %
SOR XIC I:3.0/2 OTE N11:30/2 EOR
%   I:3.0/2  "Wrap Zone "Overtravel" Is Clear" %
%   N11:30/2  WRAPZONEOVER  "- Input - Wrap Zone Overtravel Clear" %

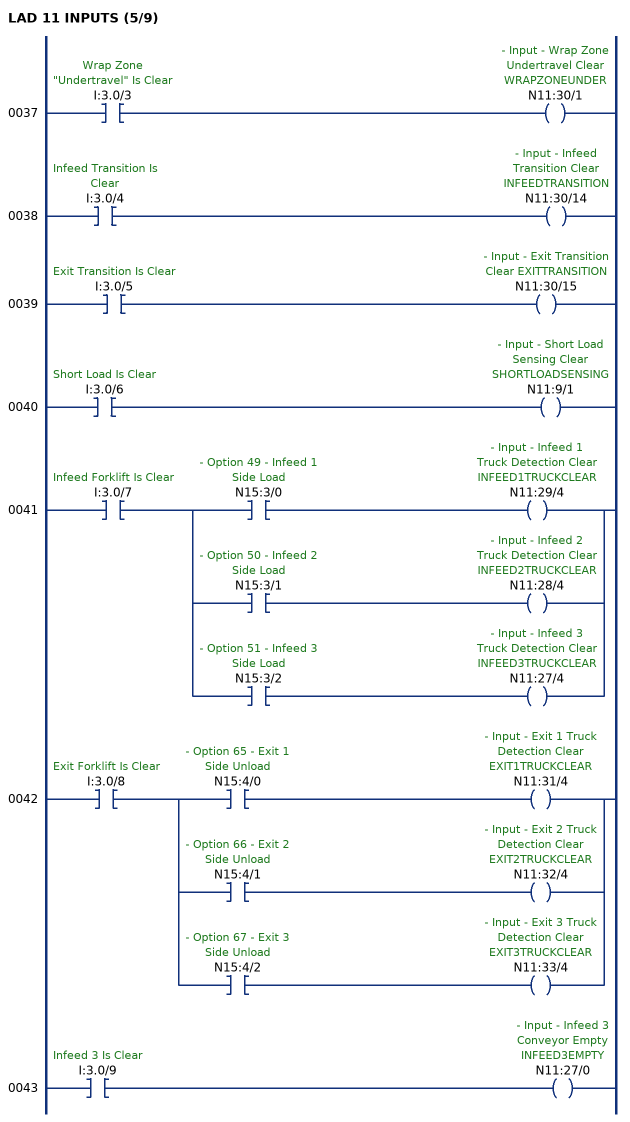
% Rung: 37 %
SOR XIC I:3.0/3 OTE N11:30/1 EOR
%   I:3.0/3  "Wrap Zone "Undertravel" Is Clear" %
%   N11:30/1  WRAPZONEUNDER  "- Input - Wrap Zone Undertravel Clear" %
% Rung: 38 %
SOR XIC I:3.0/4 OTE N11:30/14 EOR
%   I:3.0/4  "Infeed Transition Is Clear" %
%   N11:30/14  INFEEDTRANSITION  "- Input - Infeed Transition Clear" %
% Rung: 39 %
SOR XIC I:3.0/5 OTE N11:30/15 EOR
%   I:3.0/5  "Exit Transition Is Clear" %
%   N11:30/15  EXITTRANSITION  "- Input - Exit Transition Clear" %
% Rung: 40 %
SOR XIC I:3.0/6 OTE N11:9/1 EOR
%   I:3.0/6  "Short Load Is Clear" %
%   N11:9/1  SHORTLOADSENSING  "- Input - Short Load Sensing Clear" %
% Rung: 41 %
SOR XIC I:3.0/7 BST XIC N15:3/0 OTE N11:29/4 NXB XIC N15:3/1 OTE N11:28/4 NXB XIC N15:3/2 OTE N11:27/4 BND EOR
%   I:3.0/7  "Infeed Forklift Is Clear" %
%   N15:3/0  "- Option 49 - Infeed 1 Side Load" %
%   N11:29/4  INFEED1TRUCKCLEAR  "- Input - Infeed 1 Truck Detection Clear" %
%   N15:3/1  "- Option 50 - Infeed 2 Side Load" %
%   N11:28/4  INFEED2TRUCKCLEAR  "- Input - Infeed 2 Truck Detection Clear" %
%   N15:3/2  "- Option 51 - Infeed 3 Side Load" %
%   N11:27/4  INFEED3TRUCKCLEAR  "- Input - Infeed 3 Truck Detection Clear" %
% Rung: 42 %
SOR XIC I:3.0/8 BST XIC N15:4/0 OTE N11:31/4 NXB XIC N15:4/1 OTE N11:32/4 NXB XIC N15:4/2 OTE N11:33/4 BND EOR
%   I:3.0/8  "Exit Forklift Is Clear" %
%   N15:4/0  "- Option 65 - Exit 1 Side Unload" %
%   N11:31/4  EXIT1TRUCKCLEAR  "- Input - Exit 1 Truck Detection Clear" %
%   N15:4/1  "- Option 66 - Exit 2 Side Unload" %
%   N11:32/4  EXIT2TRUCKCLEAR  "- Input - Exit 2 Truck Detection Clear" %
%   N15:4/2  "- Option 67 - Exit 3 Side Unload" %
%   N11:33/4  EXIT3TRUCKCLEAR  "- Input - Exit 3 Truck Detection Clear" %
% Rung: 43 %
SOR XIC I:3.0/9 OTE N11:27/0 EOR
%   I:3.0/9  "Infeed 3 Is Clear" %
%   N11:27/0  INFEED3EMPTY  "- Input - Infeed 3 Conveyor Empty" %

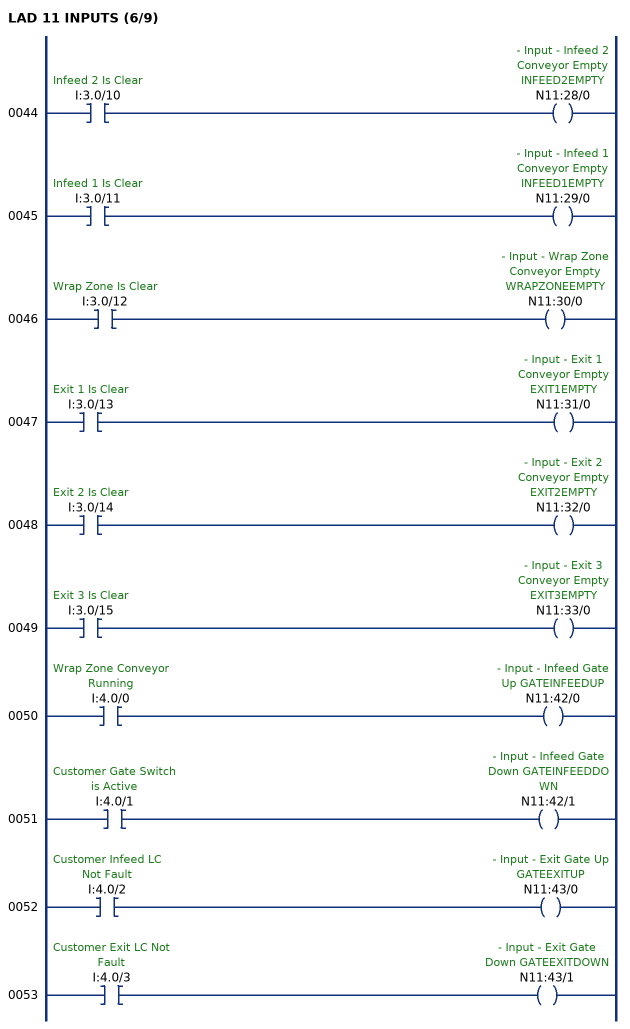
% Rung: 44 %
SOR XIC I:3.0/10 OTE N11:28/0 EOR
%   I:3.0/10  "Infeed 2 Is Clear" %
%   N11:28/0  INFEED2EMPTY  "- Input - Infeed 2 Conveyor Empty" %
% Rung: 45 %
SOR XIC I:3.0/11 OTE N11:29/0 EOR
%   I:3.0/11  "Infeed 1 Is Clear" %
%   N11:29/0  INFEED1EMPTY  "- Input - Infeed 1 Conveyor Empty" %
% Rung: 46 %
SOR XIC I:3.0/12 OTE N11:30/0 EOR
%   I:3.0/12  "Wrap Zone Is Clear" %
%   N11:30/0  WRAPZONEEMPTY  "- Input - Wrap Zone Conveyor Empty" %
% Rung: 47 %
SOR XIC I:3.0/13 OTE N11:31/0 EOR
%   I:3.0/13  "Exit 1 Is Clear" %
%   N11:31/0  EXIT1EMPTY  "- Input - Exit 1 Conveyor Empty" %
% Rung: 48 %
SOR XIC I:3.0/14 OTE N11:32/0 EOR
%   I:3.0/14  "Exit 2 Is Clear" %
%   N11:32/0  EXIT2EMPTY  "- Input - Exit 2 Conveyor Empty" %
% Rung: 49 %
SOR XIC I:3.0/15 OTE N11:33/0 EOR
%   I:3.0/15  "Exit 3 Is Clear" %
%   N11:33/0  EXIT3EMPTY  "- Input - Exit 3 Conveyor Empty" %
% Rung: 50 %
SOR XIC I:4.0/0 OTE N11:42/0 EOR
%   I:4.0/0  "Wrap Zone Conveyor Running" %
%   N11:42/0  GATEINFEEDUP  "- Input - Infeed Gate Up" %
% Rung: 51 %
SOR XIC I:4.0/1 OTE N11:42/1 EOR
%   I:4.0/1  "Customer Gate Switch is Active" %
%   N11:42/1  GATEINFEEDDOWN  "- Input - Infeed Gate Down" %
% Rung: 52 %
SOR XIC I:4.0/2 OTE N11:43/0 EOR
%   I:4.0/2  "Customer Infeed LC Not Fault" %
%   N11:43/0  GATEEXITUP  "- Input - Exit Gate Up" %
% Rung: 53 %
SOR XIC I:4.0/3 OTE N11:43/1 EOR
%   I:4.0/3  "Customer Exit LC Not Fault" %
%   N11:43/1  GATEEXITDOWN  "- Input - Exit Gate Down" %

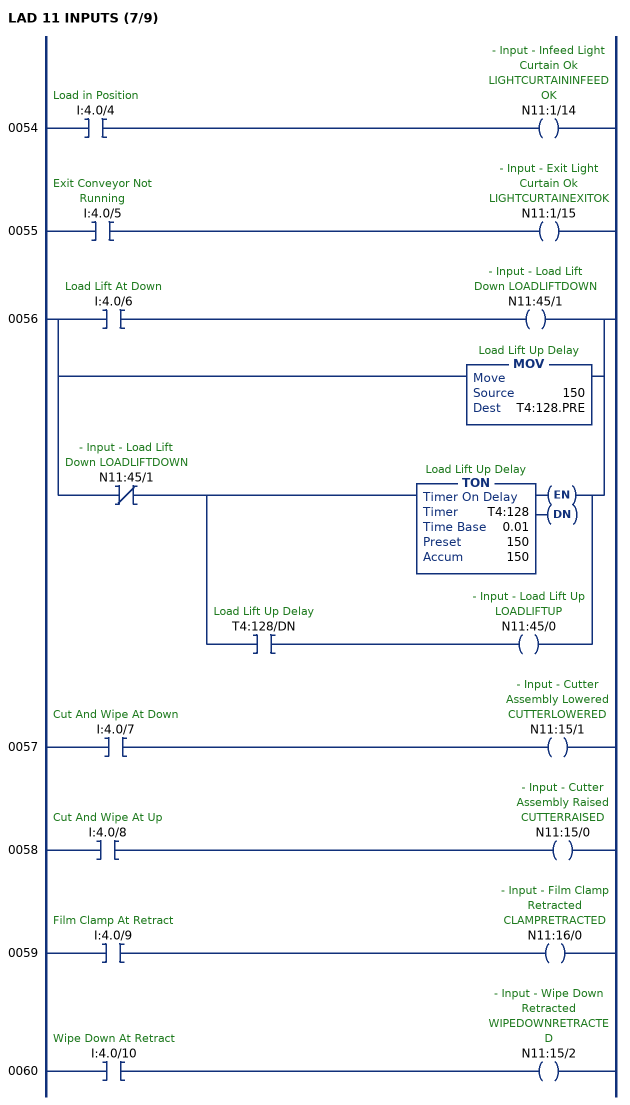
% Rung: 54 %
SOR XIC I:4.0/4 OTE N11:1/14 EOR
%   I:4.0/4  "Load in Position" %
%   N11:1/14  LIGHTCURTAININFEEDOK  "- Input - Infeed Light Curtain Ok" %
% Rung: 55 %
SOR XIC I:4.0/5 OTE N11:1/15 EOR
%   I:4.0/5  "Exit Conveyor Not Running" %
%   N11:1/15  LIGHTCURTAINEXITOK  "- Input - Exit Light Curtain Ok" %
% Rung: 56 %
SOR BST XIC I:4.0/6 OTE N11:45/1 NXB MOV 150 T4:128.PRE NXB XIO N11:45/1 BST TON T4:128 0.01 150 150 NXB XIC T4:128/DN OTE N11:45/0 BND BND EOR
%   I:4.0/6  "Load Lift At Down" %
%   N11:45/1  LOADLIFTDOWN  "- Input - Load Lift Down" %
%   T4:128  "Load Lift Up Delay" %
%   N11:45/0  LOADLIFTUP  "- Input - Load Lift Up" %
% Rung: 57 %
SOR XIC I:4.0/7 OTE N11:15/1 EOR
%   I:4.0/7  "Cut And Wipe At Down" %
%   N11:15/1  CUTTERLOWERED  "- Input - Cutter Assembly Lowered" %
% Rung: 58 %
SOR XIC I:4.0/8 OTE N11:15/0 EOR
%   I:4.0/8  "Cut And Wipe At Up" %
%   N11:15/0  CUTTERRAISED  "- Input - Cutter Assembly Raised" %
% Rung: 59 %
SOR XIC I:4.0/9 OTE N11:16/0 EOR
%   I:4.0/9  "Film Clamp At Retract" %
%   N11:16/0  CLAMPRETRACTED  "- Input - Film Clamp Retracted" %
% Rung: 60 %
SOR XIC I:4.0/10 OTE N11:15/2 EOR
%   I:4.0/10  "Wipe Down At Retract" %
%   N11:15/2  WIPEDOWNRETRACTED  "- Input - Wipe Down Retracted" %

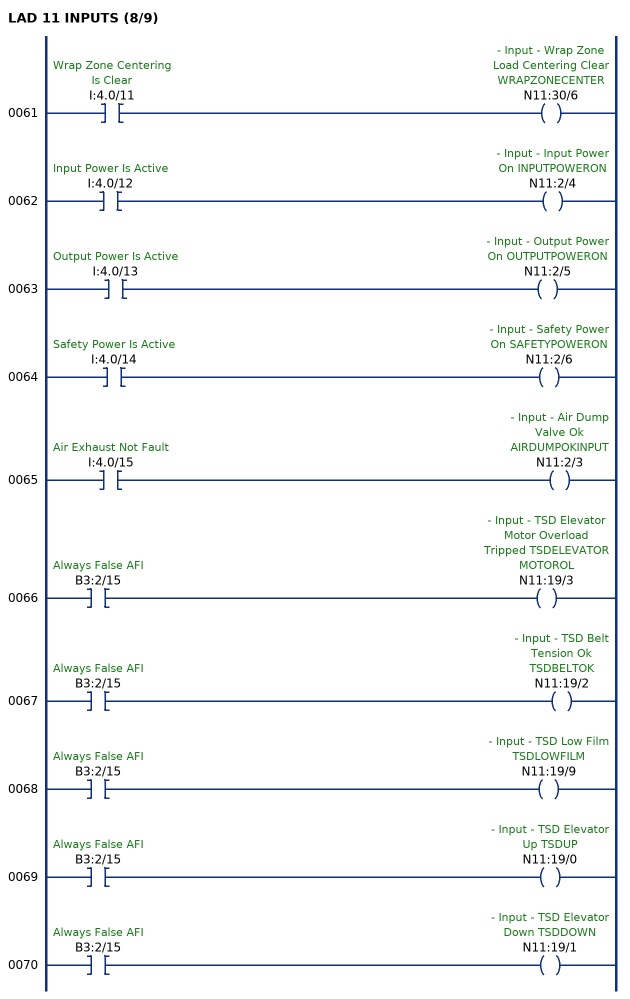
% Rung: 61 %
SOR XIC I:4.0/11 OTE N11:30/6 EOR
%   I:4.0/11  "Wrap Zone Centering Is Clear" %
%   N11:30/6  WRAPZONECENTER  "- Input - Wrap Zone Load Centering Clear" %
% Rung: 62 %
SOR XIC I:4.0/12 OTE N11:2/4 EOR
%   I:4.0/12  "Input Power Is Active" %
%   N11:2/4  INPUTPOWERON  "- Input - Input Power On" %
% Rung: 63 %
SOR XIC I:4.0/13 OTE N11:2/5 EOR
%   I:4.0/13  "Output Power Is Active" %
%   N11:2/5  OUTPUTPOWERON  "- Input - Output Power On" %
% Rung: 64 %
SOR XIC I:4.0/14 OTE N11:2/6 EOR
%   I:4.0/14  "Safety Power Is Active" %
%   N11:2/6  SAFETYPOWERON  "- Input - Safety Power On" %
% Rung: 65 %
SOR XIC I:4.0/15 OTE N11:2/3 EOR
%   I:4.0/15  "Air Exhaust Not Fault" %
%   N11:2/3  AIRDUMPOKINPUT  "- Input - Air Dump Valve Ok" %
% Rung: 66 %
SOR XIC B3:2/15 OTE N11:19/3 EOR
%   B3:2/15  AFI  "Always False" %
%   N11:19/3  TSDELEVATORMOTOROL  "- Input - TSD Elevator Motor Overload Tripped" %
% Rung: 67 %
SOR XIC B3:2/15 OTE N11:19/2 EOR
%   B3:2/15  AFI  "Always False" %
%   N11:19/2  TSDBELTOK  "- Input - TSD Belt Tension Ok" %
% Rung: 68 %
SOR XIC B3:2/15 OTE N11:19/9 EOR
%   B3:2/15  AFI  "Always False" %
%   N11:19/9  TSDLOWFILM  "- Input - TSD Low Film" %
% Rung: 69 %
SOR XIC B3:2/15 OTE N11:19/0 EOR
%   B3:2/15  AFI  "Always False" %
%   N11:19/0  TSDUP  "- Input - TSD Elevator Up" %
% Rung: 70 %
SOR XIC B3:2/15 OTE N11:19/1 EOR
%   B3:2/15  AFI  "Always False" %
%   N11:19/1  TSDDOWN  "- Input - TSD Elevator Down" %

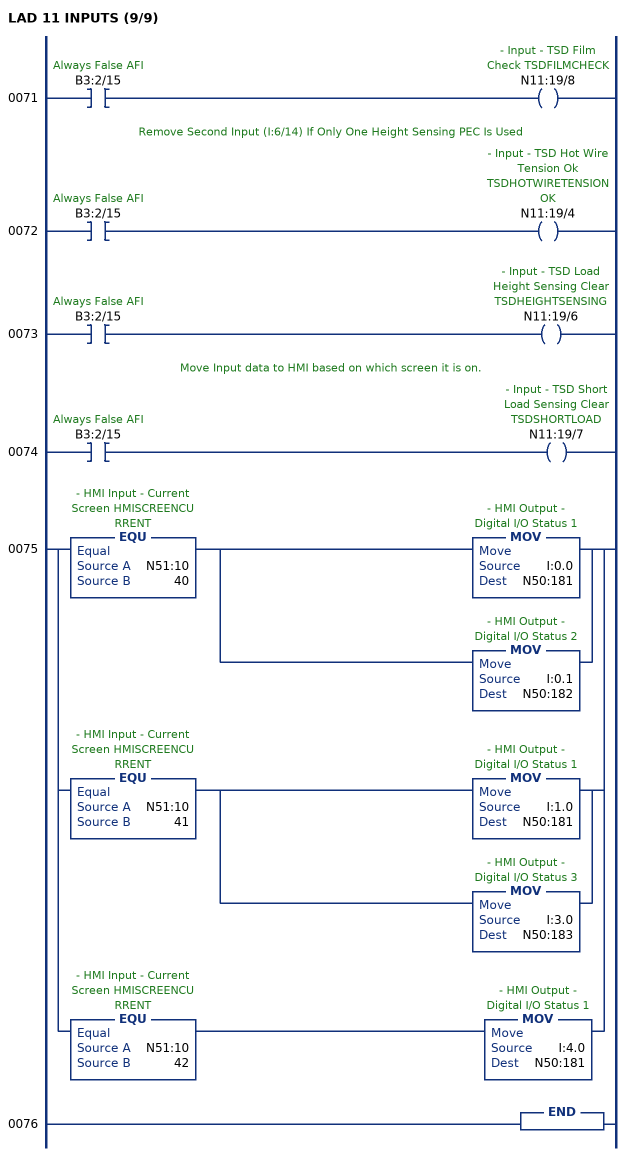
% Rung: 71 %
SOR XIC B3:2/15 OTE N11:19/8 EOR
%   B3:2/15  AFI  "Always False" %
%   N11:19/8  TSDFILMCHECK  "- Input - TSD Film Check" %
% Rung: 72 %
% Remove Second Input (I:6/14) If Only One Height Sensing PEC Is Used %
SOR XIC B3:2/15 OTE N11:19/4 EOR
%   B3:2/15  AFI  "Always False" %
%   N11:19/4  TSDHOTWIRETENSIONOK  "- Input - TSD Hot Wire Tension Ok" %
% Rung: 73 %
SOR XIC B3:2/15 OTE N11:19/6 EOR
%   B3:2/15  AFI  "Always False" %
%   N11:19/6  TSDHEIGHTSENSING  "- Input - TSD Load Height Sensing Clear" %
% Rung: 74 %
% Move Input data to HMI based on which screen it is on. %
SOR XIC B3:2/15 OTE N11:19/7 EOR
%   B3:2/15  AFI  "Always False" %
%   N11:19/7  TSDSHORTLOAD  "- Input - TSD Short Load Sensing Clear" %
% Rung: 75 %
SOR BST EQU N51:10 40 BST MOV I:0.0 N50:181 NXB MOV I:0.1 N50:182 BND NXB EQU N51:10 41 BST MOV I:1.0 N50:181 NXB MOV I:3.0 N50:183 BND NXB EQU N51:10 42 MOV I:4.0 N50:181 BND EOR
%   N51:10  HMISCREENCURRENT  "- HMI Input - Current Screen" %
%   N50:181  "- HMI Output - Digital I/O Status 1" %
%   N50:182  "- HMI Output - Digital I/O Status 2" %
%   N50:183  "- HMI Output - Digital I/O Status 3" %
% Rung: 76 %
SOR END EOR

LADDER 12 "ROTATION"
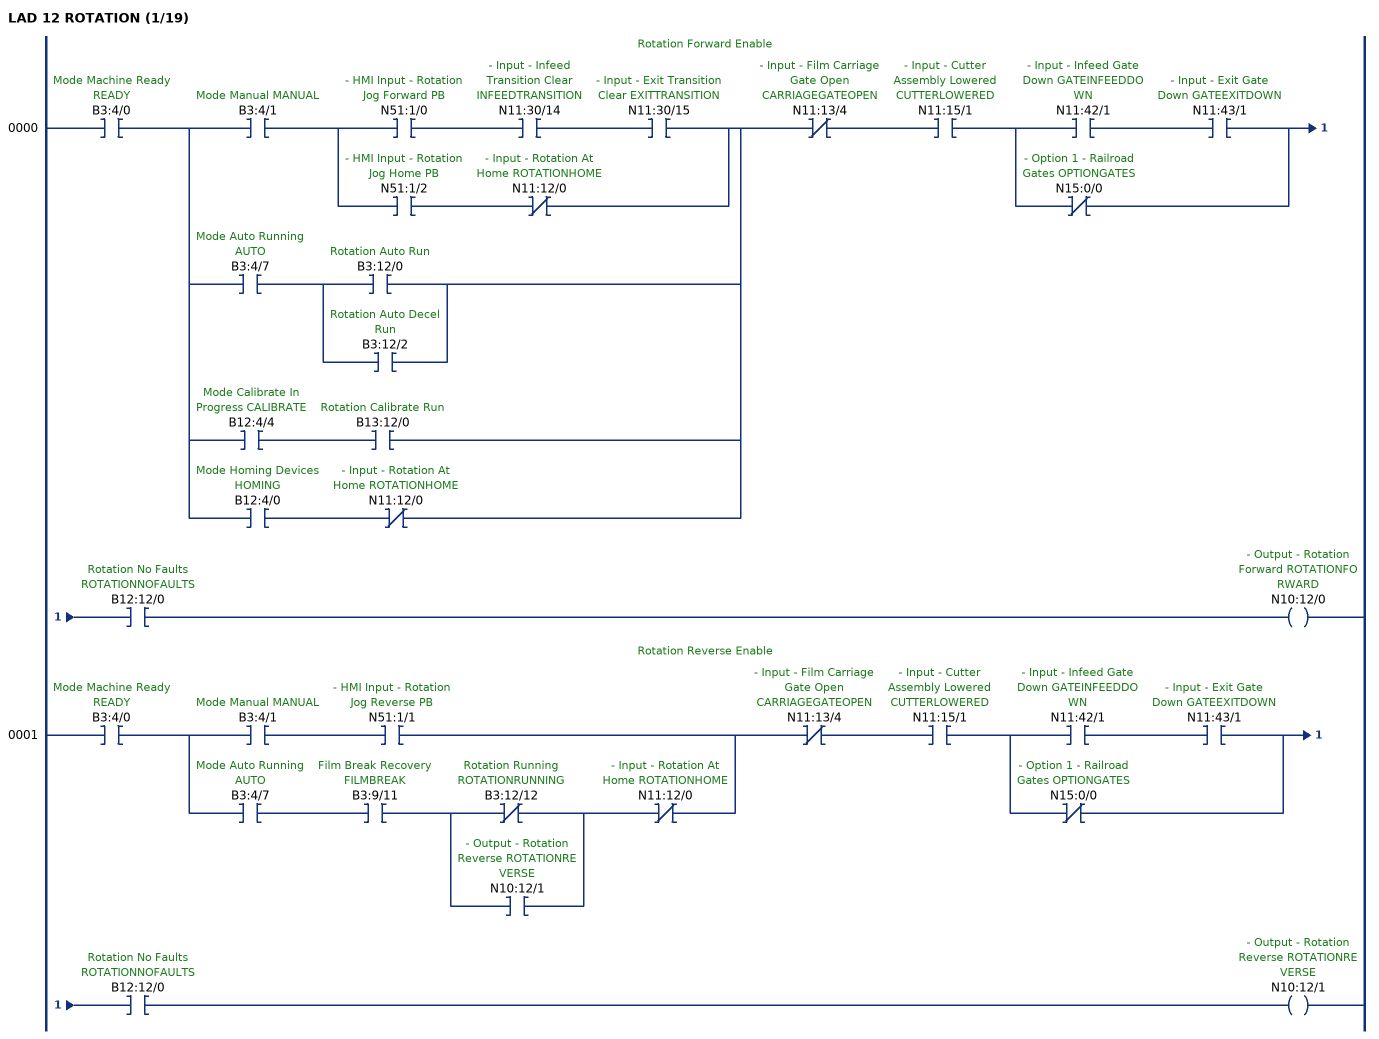
% Rung: 0 %
% Rotation Forward Enable %
SOR XIC B3:4/0 BST XIC B3:4/1 BST XIC N51:1/0 XIC N11:30/14 XIC N11:30/15 NXB XIC N51:1/2 XIO N11:12/0 BND NXB XIC B3:4/7 BST XIC B3:12/0 NXB XIC B3:12/2 BND NXB XIC B12:4/4 XIC B13:12/0 NXB XIC B12:4/0 XIO N11:12/0 BND XIO N11:13/4 XIC N11:15/1 BST XIC N11:42/1 XIC N11:43/1 NXB XIO N15:0/0 BND XIC B12:12/0 OTE N10:12/0 EOR
%   B3:4/0  READY  "Mode Machine Ready" %
%   B3:4/1  MANUAL  "Mode Manual" %
%   N51:1/0  "- HMI Input - Rotation Jog Forward PB" %
%   N11:30/14  INFEEDTRANSITION  "- Input - Infeed Transition Clear" %
%   N11:30/15  EXITTRANSITION  "- Input - Exit Transition Clear" %
%   N51:1/2  "- HMI Input - Rotation Jog Home PB" %
%   N11:12/0  ROTATIONHOME  "- Input - Rotation At Home" %
%   B3:4/7  AUTO  "Mode Auto Running" %
%   B3:12/0  "Rotation Auto Run" %
%   B3:12/2  "Rotation Auto Decel Run" %
%   B12:4/4  CALIBRATE  "Mode Calibrate In Progress" %
%   B13:12/0  "Rotation Calibrate Run" %
%   B12:4/0  HOMING  "Mode Homing Devices" %
%   N11:13/4  CARRIAGEGATEOPEN  "- Input - Film Carriage Gate Open" %
%   N11:15/1  CUTTERLOWERED  "- Input - Cutter Assembly Lowered" %
%   N11:42/1  GATEINFEEDDOWN  "- Input - Infeed Gate Down" %
%   N11:43/1  GATEEXITDOWN  "- Input - Exit Gate Down" %
%   N15:0/0  OPTIONGATES  "- Option 1 - Railroad Gates" %
%   B12:12/0  ROTATIONNOFAULTS  "Rotation No Faults" %
%   N10:12/0  ROTATIONFORWARD  "- Output - Rotation Forward" %
% Rung: 1 %
% Rotation Reverse Enable %
SOR XIC B3:4/0 BST XIC B3:4/1 XIC N51:1/1 NXB XIC B3:4/7 XIC B3:9/11 BST XIO B3:12/12 NXB XIC N10:12/1 BND XIO N11:12/0 BND XIO N11:13/4 XIC N11:15/1 BST XIC N11:42/1 XIC N11:43/1 NXB XIO N15:0/0 BND XIC B12:12/0 OTE N10:12/1 EOR
%   B3:4/0  READY  "Mode Machine Ready" %
%   B3:4/1  MANUAL  "Mode Manual" %
%   N51:1/1  "- HMI Input - Rotation Jog Reverse PB" %
%   B3:4/7  AUTO  "Mode Auto Running" %
%   B3:9/11  FILMBREAK  "Film Break Recovery" %
%   B3:12/12  ROTATIONRUNNING  "Rotation Running" %
%   N10:12/1  ROTATIONREVERSE  "- Output - Rotation Reverse" %
%   N11:12/0  ROTATIONHOME  "- Input - Rotation At Home" %
%   N11:13/4  CARRIAGEGATEOPEN  "- Input - Film Carriage Gate Open" %
%   N11:15/1  CUTTERLOWERED  "- Input - Cutter Assembly Lowered" %
%   N11:42/1  GATEINFEEDDOWN  "- Input - Infeed Gate Down" %
%   N11:43/1  GATEEXITDOWN  "- Input - Exit Gate Down" %
%   N15:0/0  OPTIONGATES  "- Option 1 - Railroad Gates" %
%   B12:12/0  ROTATIONNOFAULTS  "Rotation No Faults" %

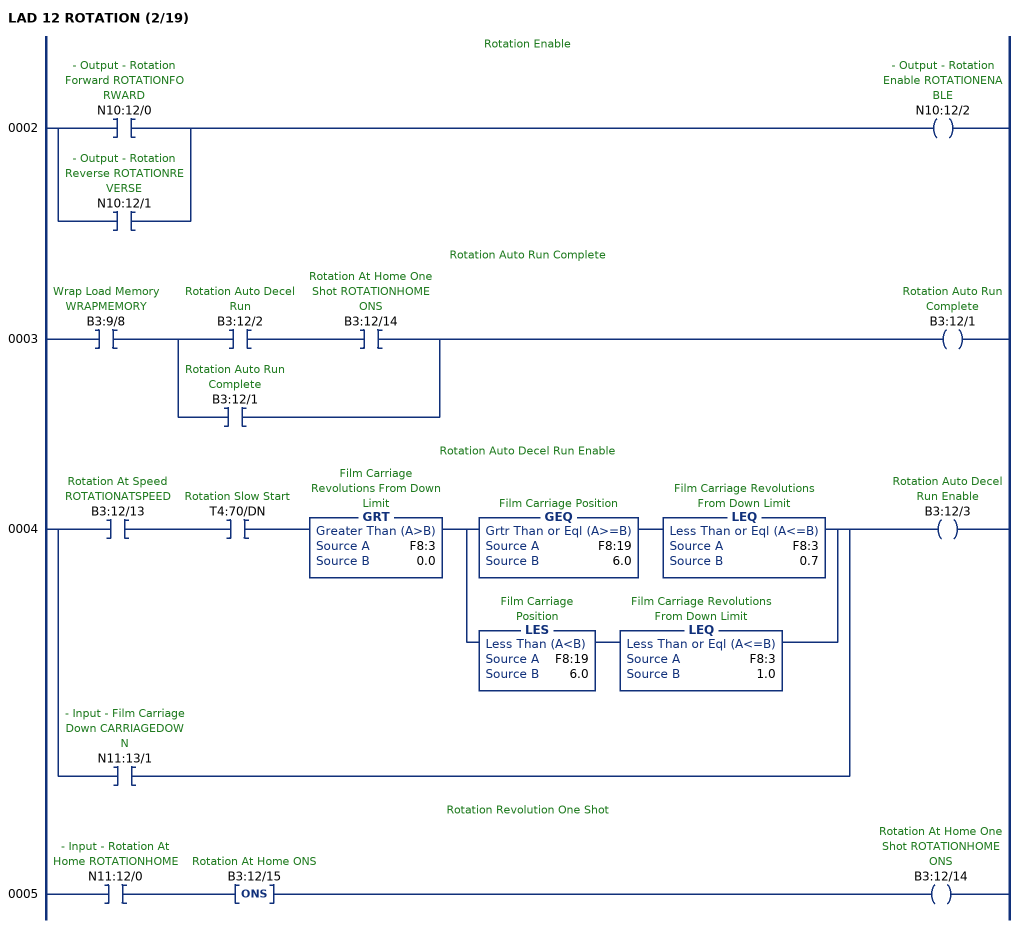
% Rung: 2 %
% Rotation Enable %
SOR BST XIC N10:12/0 NXB XIC N10:12/1 BND OTE N10:12/2 EOR
%   N10:12/0  ROTATIONFORWARD  "- Output - Rotation Forward" %
%   N10:12/1  ROTATIONREVERSE  "- Output - Rotation Reverse" %
%   N10:12/2  ROTATIONENABLE  "- Output - Rotation Enable" %
% Rung: 3 %
% Rotation Auto Run Complete %
SOR XIC B3:9/8 BST XIC B3:12/2 XIC B3:12/14 NXB XIC B3:12/1 BND OTE B3:12/1 EOR
%   B3:9/8  WRAPMEMORY  "Wrap Load Memory" %
%   B3:12/2  "Rotation Auto Decel Run" %
%   B3:12/14  ROTATIONHOMEONS  "Rotation At Home One Shot" %
%   B3:12/1  "Rotation Auto Run Complete" %
% Rung: 4 %
% Rotation Auto Decel Run Enable %
SOR BST XIC B3:12/13 XIC T4:70/DN GRT F8:3 0.0 BST GEQ F8:19 6.0 LEQ F8:3 0.7 NXB LES F8:19 6.0 LEQ F8:3 1.0 BND NXB XIC N11:13/1 BND OTE B3:12/3 EOR
%   B3:12/13  ROTATIONATSPEED  "Rotation At Speed" %
%   T4:70  "Rotation Slow Start" %
%   F8:3  "Film Carriage Revolutions From Down Limit" %
%   F8:19  "Film Carriage Position" %
%   N11:13/1  CARRIAGEDOWN  "- Input - Film Carriage Down" %
%   B3:12/3  "Rotation Auto Decel Run Enable" %
% Rung: 5 %
% Rotation Revolution One Shot %
SOR XIC N11:12/0 ONS B3:12/15 OTE B3:12/14 EOR
%   N11:12/0  ROTATIONHOME  "- Input - Rotation At Home" %
%   B3:12/15  "Rotation At Home ONS" %
%   B3:12/14  ROTATIONHOMEONS  "Rotation At Home One Shot" %

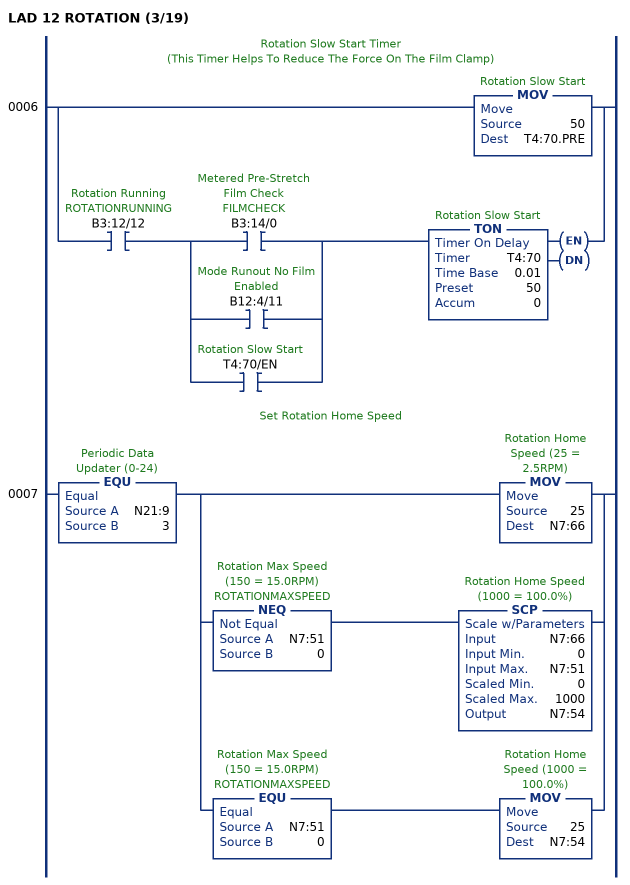
% Rung: 6 %
% Rotation Slow Start Timer
% (This Timer Helps To Reduce The Force On The Film Clamp) %
SOR BST MOV 50 T4:70.PRE NXB XIC B3:12/12 BST XIC B3:14/0 NXB XIC B12:4/11 NXB XIC T4:70/EN BND TON T4:70 0.01 50 0 BND EOR
%   T4:70  "Rotation Slow Start" %
%   B3:12/12  ROTATIONRUNNING  "Rotation Running" %
%   B3:14/0  FILMCHECK  "Metered Pre-Stretch Film Check" %
%   B12:4/11  "Mode Runout No Film Enabled" %
% Rung: 7 %
% Set Rotation Home Speed %
SOR EQU N21:9 3 BST MOV 25 N7:66 NXB NEQ N7:51 0 SCP N7:66 0 N7:51 0 1000 N7:54 NXB EQU N7:51 0 MOV 25 N7:54 BND EOR
%   N21:9  "Periodic Data Updater (0-24)" %
%   N7:66  "Rotation Home Speed (25 = 2.5RPM)" %
%   N7:51  ROTATIONMAXSPEED  "Rotation Max Speed (150 = 15.0RPM)" %
%   N7:54  "Rotation Home Speed (1000 = 100.0%)" %

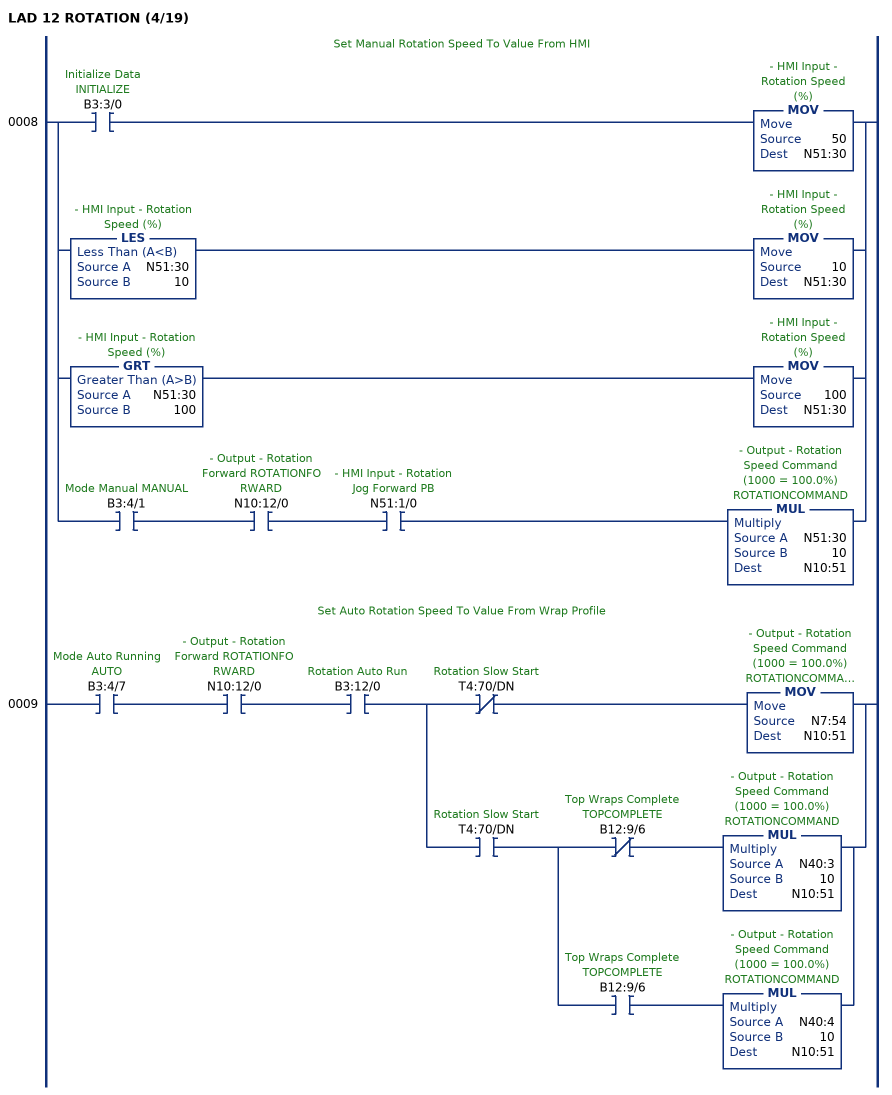
% Rung: 8 %
% Set Manual Rotation Speed To Value From HMI %
SOR BST BST XIC B3:3/0 MOV 50 N51:30 NXB LES N51:30 10 MOV 10 N51:30 NXB GRT N51:30 100 MOV 100 N51:30 BND NXB XIC B3:4/1 XIC N10:12/0 XIC N51:1/0 MUL N51:30 10 N10:51 BND EOR
%   B3:3/0  INITIALIZE  "Initialize Data" %
%   N51:30  "- HMI Input - Rotation Speed (%)" %
%   B3:4/1  MANUAL  "Mode Manual" %
%   N10:12/0  ROTATIONFORWARD  "- Output - Rotation Forward" %
%   N51:1/0  "- HMI Input - Rotation Jog Forward PB" %
%   N10:51  ROTATIONCOMMAND  "- Output - Rotation Speed Command (1000 = 100.0%)" %
% Rung: 9 %
% Set Auto Rotation Speed To Value From Wrap Profile %
SOR XIC B3:4/7 XIC N10:12/0 XIC B3:12/0 BST XIO T4:70/DN MOV N7:54 N10:51 NXB XIC T4:70/DN BST XIO B12:9/6 MUL N40:3 10 N10:51 NXB XIC B12:9/6 MUL N40:4 10 N10:51 BND BND EOR
%   B3:4/7  AUTO  "Mode Auto Running" %
%   N10:12/0  ROTATIONFORWARD  "- Output - Rotation Forward" %
%   B3:12/0  "Rotation Auto Run" %
%   T4:70  "Rotation Slow Start" %
%   N7:54  "Rotation Home Speed (1000 = 100.0%)" %
%   N10:51  ROTATIONCOMMAND  "- Output - Rotation Speed Command (1000 = 100.0%)" %
%   B12:9/6  TOPCOMPLETE  "Top Wraps Complete" %
%   N40:3  "Current Profile Rotation Up Speed (%)" %
%   N40:4  "Current Profile Rotation Down Speed (%)" %

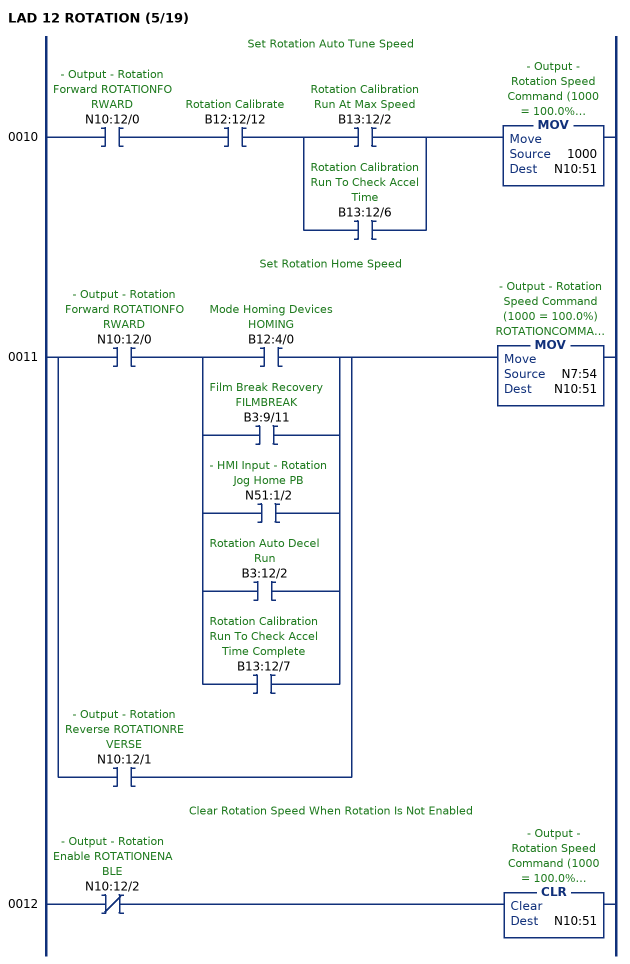
% Rung: 10 %
% Set Rotation Auto Tune Speed %
SOR XIC N10:12/0 XIC B12:12/12 BST XIC B13:12/2 NXB XIC B13:12/6 BND MOV 1000 N10:51 EOR
%   N10:12/0  ROTATIONFORWARD  "- Output - Rotation Forward" %
%   B12:12/12  "Rotation Calibrate" %
%   B13:12/2  "Rotation Calibration Run At Max Speed" %
%   B13:12/6  "Rotation Calibration Run To Check Accel Time" %
%   N10:51  ROTATIONCOMMAND  "- Output - Rotation Speed Command (1000 = 100.0%)" %
% Rung: 11 %
% Set Rotation Home Speed %
SOR BST XIC N10:12/0 BST XIC B12:4/0 NXB XIC B3:9/11 NXB XIC N51:1/2 NXB XIC B3:12/2 NXB XIC B13:12/7 BND NXB XIC N10:12/1 BND MOV N7:54 N10:51 EOR
%   N10:12/0  ROTATIONFORWARD  "- Output - Rotation Forward" %
%   B12:4/0  HOMING  "Mode Homing Devices" %
%   B3:9/11  FILMBREAK  "Film Break Recovery" %
%   N51:1/2  "- HMI Input - Rotation Jog Home PB" %
%   B3:12/2  "Rotation Auto Decel Run" %
%   B13:12/7  "Rotation Calibration Run To Check Accel Time Complete" %
%   N10:12/1  ROTATIONREVERSE  "- Output - Rotation Reverse" %
%   N7:54  "Rotation Home Speed (1000 = 100.0%)" %
%   N10:51  ROTATIONCOMMAND  "- Output - Rotation Speed Command (1000 = 100.0%)" %
% Rung: 12 %
% Clear Rotation Speed When Rotation Is Not Enabled %
SOR XIO N10:12/2 CLR N10:51 EOR
%   N10:12/2  ROTATIONENABLE  "- Output - Rotation Enable" %
%   N10:51  ROTATIONCOMMAND  "- Output - Rotation Speed Command (1000 = 100.0%)" %

